KUKA KRL program: EPS_2_25716_MHCR11_A_20250905053025.src

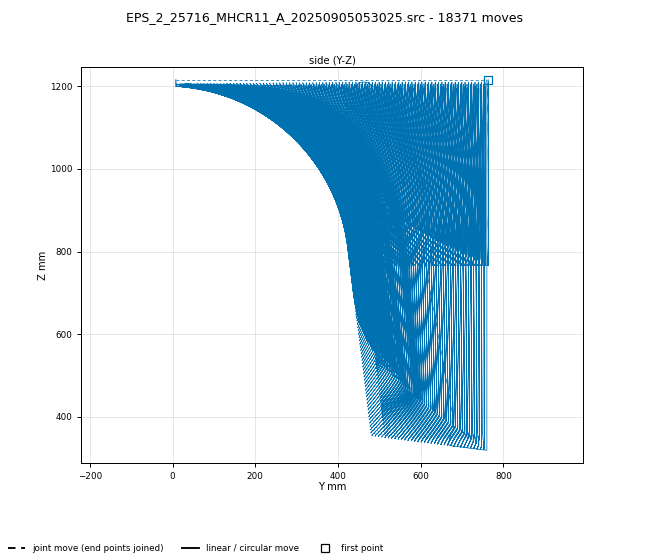
[picture p0: tool path of EPS_2_25716_MHCR11_A_20250905053025.src, 18371 of 18373 moves have a stored position in this frame; points joined in program order, loops and branches not executed]
&ACCESS RVP
&REL 4
&COMMENT QRS 19112012
&PARAM EDITMASK = *
DEF PART()
EXT BAS (BAS_COMMAND :IN,REAL :IN )
INT I
BAS (#INITMOV,0 )

;KUKA QRS Post kuka4.cps  Date:22-06-2017 !

File_ID=2809

QRS_PRE_INIT()

;Init var - Until changes are made in qrs_pre_init
Outlet_Square_prg=0
Inlet_1_Square_prg=0
Inlet_2_Square_prg=0
Inlet_3_Square_prg=0
Inlet_4_Square_prg=0
Inlet_5_Square_prg=0

Outlet_1={X 0.000, Y 457.000, Z 786.000, B 0.000, E1 0.000 }
Inlet_1={X 0.000, Y 457.000, Z 776.000, B 0.000, E1 174.000 }
Outlet_1_type=838
Inlet_1_type=838
;QRS#1=Sidecore dimensions
;QRS#2=825-33" Concrete
;QRS#3=825-33" Concrete
;QRS#4=
;QRS#5=
;QRS#6=
;QRS#7=
;QRS#8=
;QRS#9=S306-46
;QRS#10=S306-46
;QRS#11=
;QRS#12=
;QRS#13=
;QRS#14=
;QRS#15=
;QRS#16=1524x152x1676 5,5'
;QRS#17=EPS Height
;QRS#18=1205
;QRS#19=*
;QRS#20= UPDATED VERSION 22-06-2017
;QRS#21=*
Outlet_Square=0650
Inlet_1_Square=0650
Inlet_2_Square=0
Inlet_3_Square=0
Inlet_4_Square=0
Inlet_5_Square=0
Mill_Square=1
Outlet_Square_Prg=267
Inlet_1_Square_prg=267

QRS_INIT()

$ADVANCE=5

; T1
PTP {E1 176.625,E2 176.625}
PTP {X 0,Y 763.403,A -85,B 0,C 180,E1 176.625,E2 176.625,E3 0,E4 0,E5 0,E6 0}
QRS_SPEED_INIT()
LIN {X 0,Y 763.403,Z 1215,A -85,B 0,C 180,E1 176.625,E2 176.625,E3 0,E4 0,E5 0,E6 0} C_VEL
LIN {X 0,Y 763.403,Z 769.06,A -85,B 0,C 180,E1 176.625,E2 176.625} C_VEL
LIN {X 0,Y 763.516,Z 767.06,A -85,B 0,C 180,E1 176.775,E2 176.775} C_VEL
LIN {X 0,Y 763.851,Z 767.06,A -85,B 0,C 180,E1 177.187,E2 177.187} C_VEL
LIN {X 0,Y 763.775,Z 767.06,A -85,B 0,C 180,E1 184.693,E2 184.693} C_VEL
LIN {X 0,Y 763.789,Z 767.06,A -85,B 0,C 180,E1 192.281,E2 192.281} C_VEL
LIN {X 0,Y 763.833,Z 767.06,A -85,B 0,C 180,E1 200.095,E2 200.095} C_VEL
LIN {X 0,Y 763.8,Z 767.06,A -85,B 0,C 180,E1 208.326,E2 208.326} C_VEL
LIN {X 0,Y 762.389,Z 767.06,A -85,B 0,C 180,E1 210.541,E2 210.541} C_VEL
LIN {X 0,Y 762.703,Z 767.06,A -85,B 0,C 180,E1 214.993,E2 214.993} C_VEL
LIN {X 0,Y 763.704,Z 767.06,A -85,B 0,C 180,E1 216.697,E2 216.697} C_VEL
LIN {X 0,Y 763.451,Z 767.06,A -85,B 0,C 180,E1 224.739,E2 224.739} C_VEL
LIN {X 0,Y 763.703,Z 767.06,A -85,B 0,C 180,E1 225.281,E2 225.281} C_VEL
LIN {X 0,Y 763.812,Z 767.06,A -85,B 0,C 180,E1 233.406,E2 233.406} C_VEL
LIN {X 0,Y 763.419,Z 767.06,A -85,B 0,C 180,E1 233.624,E2 233.624} C_VEL
LIN {X 0,Y 763.046,Z 767.06,A -85,B 0,C 180,E1 233.668,E2 233.668} C_VEL
LIN {X 0,Y 762.775,Z 769.023,A -85,B 0,C 180,E1 233.717,E2 233.717} C_VEL
LIN {X 0,Y 763.466,Z 807.779,A -85,B 0,C 180,E1 234.197,E2 234.197} C_VEL
LIN {X 0,Y 763.742,Z 829.636,A -85,B 0,C 180,E1 234.483,E2 234.483} C_VEL
LIN {X 0,Y 763.754,Z 846.275,A -85,B 0,C 180,E1 234.748,E2 234.748} C_VEL
LIN {X 0,Y 763.618,Z 862.338,A -85,B 0,C 180,E1 235.056,E2 235.056} C_VEL
LIN {X 0,Y 763.237,Z 876.777,A -85,B 0,C 180,E1 235.362,E2 235.362} C_VEL
LIN {X 0,Y 763.626,Z 894.422,A -85,B 0,C 180,E1 235.847,E2 235.847} C_VEL
LIN {X 0,Y 763.699,Z 916.902,A -85,B 0,C 180,E1 236.542,E2 236.542} C_VEL
LIN {X 0,Y 763.604,Z 937.208,A -85,B 0,C 180,E1 237.264,E2 237.264} C_VEL
LIN {X 0,Y 763.43,Z 948.906,A -85,B 0,C 180,E1 237.721,E2 237.721} C_VEL
LIN {X 0,Y 763.574,Z 957.186,A -85,B 0,C 180,E1 238.074,E2 238.074} C_VEL
LIN {X 0,Y 763.561,Z 973.321,A -85,B 0,C 180,E1 238.795,E2 238.795} C_VEL
LIN {X 0,Y 763.553,Z 990.951,A -85,B 0,C 180,E1 239.666,E2 239.666} C_VEL
LIN {X 0,Y 763.64,Z 1008.434,A -85,B 0,C 180,E1 240.621,E2 240.621} C_VEL
LIN {X 0,Y 763.573,Z 1024.267,A -85,B 0,C 180,E1 241.555,E2 241.555} C_VEL
LIN {X 0,Y 763.324,Z 1040.379,A -85,B 0,C 180,E1 242.584,E2 242.584} C_VEL
LIN {X 0,Y 763.281,Z 1055.421,A -85,B 0,C 180,E1 243.634,E2 243.634} C_VEL
LIN {X 0,Y 763.581,Z 1070.933,A -85,B 0,C 180,E1 244.825,E2 244.825} C_VEL
LIN {X 0,Y 763.679,Z 1081.725,A -85,B 0,C 180,E1 245.706,E2 245.706} C_VEL
LIN {X 0,Y 763.252,Z 1096.523,A -85,B 0,C 180,E1 246.989,E2 246.989} C_VEL
LIN {X 0,Y 763.129,Z 1109.853,A -85,B 0,C 180,E1 248.262,E2 248.262} C_VEL
LIN {X 0,Y 763.47,Z 1121.627,A -85,B 0,C 180,E1 249.493,E2 249.493} C_VEL
LIN {X 0,Y 763.789,Z 1128.839,A -85,B 0,C 180,E1 250.312,E2 250.312} C_VEL
LIN {X 0,Y 763.599,Z 1133.682,A -85,B 0,C 180,E1 250.86,E2 250.86} C_VEL
LIN {X 0,Y 763.002,Z 1144.009,A -85,B 0,C 180,E1 252.116,E2 252.116} C_VEL
LIN {X 0,Y 762.888,Z 1154.837,A -85,B 0,C 180,E1 253.587,E2 253.587} C_VEL
LIN {X 0,Y 763.437,Z 1163.995,A -85,B 0,C 180,E1 254.972,E2 254.972} C_VEL
LIN {X 0,Y 763.849,Z 1168.884,A -85,B 0,C 180,E1 255.795,E2 255.795} C_VEL
LIN {X 0,Y 763.459,Z 1172.713,A -85,B 0,C 180,E1 256.432,E2 256.432} C_VEL
LIN {X 0,Y 762.709,Z 1180.75,A -85,B 0,C 180,E1 257.942,E2 257.942} C_VEL
LIN {X 0,Y 762.709,Z 1187.417,A -85,B 0,C 180,E1 259.378,E2 259.378} C_VEL
LIN {X 0,Y 763.283,Z 1192.233,A -85,B 0,C 180,E1 260.577,E2 260.577} C_VEL
LIN {X 0,Y 763.861,Z 1195.667,A -85,B 0,C 180,E1 261.533,E2 261.533} C_VEL
LIN {X 0,Y 763.274,Z 1198.713,A -85,B 0,C 180,E1 262.474,E2 262.474} C_VEL
LIN {X 0,Y 762.669,Z 1202.591,A -85,B 0,C 180,E1 263.886,E2 263.886} C_VEL
LIN {X 0,Y 762.823,Z 1205.612,A -85,B 0,C 180,E1 265.302,E2 265.302} C_VEL
LIN {X 0,Y 763.582,Z 1207.795,A -85,B 0,C 180,E1 266.708,E2 266.708} C_VEL
LIN {X 0,Y 763.887,Z 1208.357,A -85,B 0,C 180,E1 267.187,E2 267.187} C_VEL
LIN {X 0,Y 762.685,Z 1209.719,A -85,B 0,C 180,E1 269.062,E2 269.062} C_VEL
LIN {X 0,Y 762.503,Z 1209.722,A -85,B 0,C 180,E1 270.939,E2 270.939} C_VEL
LIN {X 0,Y 763.555,Z 1208.375,A -85,B 0,C 180,E1 272.815,E2 272.815} C_VEL
LIN {X 0,Y 763.68,Z 1207.369,A -85,B 0,C 180,E1 273.603,E2 273.603} C_VEL
LIN {X 0,Y 763.024,Z 1205.607,A -85,B 0,C 180,E1 274.698,E2 274.698} C_VEL
LIN {X 0,Y 762.624,Z 1202.589,A -85,B 0,C 180,E1 276.115,E2 276.115} C_VEL
LIN {X 0,Y 763.008,Z 1198.714,A -85,B 0,C 180,E1 277.529,E2 277.529} C_VEL
LIN {X 0,Y 763.565,Z 1195.67,A -85,B 0,C 180,E1 278.471,E2 278.471} C_VEL
LIN {X 0,Y 763.861,Z 1193.987,A -85,B 0,C 180,E1 278.942,E2 278.942} C_VEL
LIN {X 0,Y 763.295,Z 1190.396,A -85,B 0,C 180,E1 279.899,E2 279.899} C_VEL
LIN {X 0,Y 762.849,Z 1186.331,A -85,B 0,C 180,E1 280.859,E2 280.859} C_VEL
LIN {X 0,Y 762.72,Z 1179.546,A -85,B 0,C 180,E1 282.299,E2 282.299} C_VEL
LIN {X 0,Y 763.241,Z 1172.709,A -85,B 0,C 180,E1 283.573,E2 283.573} C_VEL
LIN {X 0,Y 763.817,Z 1166.178,A -85,B 0,C 180,E1 284.656,E2 284.656} C_VEL
LIN {X 0,Y 763.575,Z 1163.464,A -85,B 0,C 180,E1 285.111,E2 285.111} C_VEL
LIN {X 0,Y 762.944,Z 1153.1,A -85,B 0,C 180,E1 286.658,E2 286.658} C_VEL
LIN {X 0,Y 762.95,Z 1144.002,A -85,B 0,C 180,E1 287.886,E2 287.886} C_VEL
LIN {X 0,Y 763.507,Z 1132.817,A -85,B 0,C 180,E1 289.248,E2 289.248} C_VEL
LIN {X 0,Y 763.777,Z 1127.109,A -85,B 0,C 180,E1 289.882,E2 289.882} C_VEL
LIN {X 0,Y 763.473,Z 1119.599,A -85,B 0,C 180,E1 290.721,E2 290.721} C_VEL
LIN {X 0,Y 763.074,Z 1107.203,A -85,B 0,C 180,E1 292,E2 292} C_VEL
LIN {X 0,Y 763.142,Z 1095.102,A -85,B 0,C 180,E1 293.143,E2 293.143} C_VEL
LIN {X 0,Y 763.577,Z 1080.937,A -85,B 0,C 180,E1 294.361,E2 294.361} C_VEL
LIN {X 0,Y 763.638,Z 1069.815,A -85,B 0,C 180,E1 295.264,E2 295.264} C_VEL
LIN {X 0,Y 763.313,Z 1053.595,A -85,B 0,C 180,E1 296.496,E2 296.496} C_VEL
LIN {X 0,Y 763.281,Z 1038.391,A -85,B 0,C 180,E1 297.551,E2 297.551} C_VEL
LIN {X 0,Y 763.531,Z 1021.454,A -85,B 0,C 180,E1 298.617,E2 298.617} C_VEL
LIN {X 0,Y 763.61,Z 1005.589,A -85,B 0,C 180,E1 299.542,E2 299.542} C_VEL
LIN {X 0,Y 763.569,Z 987.905,A -85,B 0,C 180,E1 300.489,E2 300.489} C_VEL
LIN {X 0,Y 763.539,Z 970.163,A -85,B 0,C 180,E1 301.353,E2 301.353} C_VEL
LIN {X 0,Y 763.605,Z 952.774,A -85,B 0,C 180,E1 302.117,E2 302.117} C_VEL
LIN {X 0,Y 763.432,Z 938.395,A -85,B 0,C 180,E1 302.697,E2 302.697} C_VEL
LIN {X 0,Y 763.616,Z 929.2,A -85,B 0,C 180,E1 303.028,E2 303.028} C_VEL
LIN {X 0,Y 763.715,Z 913.957,A -85,B 0,C 180,E1 303.553,E2 303.553} C_VEL
LIN {X 0,Y 763.679,Z 893.472,A -85,B 0,C 180,E1 304.176,E2 304.176} C_VEL
LIN {X 0,Y 763.499,Z 875.748,A -85,B 0,C 180,E1 304.649,E2 304.649} C_VEL
LIN {X 0,Y 763.243,Z 865.606,A -85,B 0,C 180,E1 304.895,E2 304.895} C_VEL
LIN {X 0,Y 763.621,Z 848.959,A -85,B 0,C 180,E1 305.209,E2 305.209} C_VEL
LIN {X 0,Y 763.7,Z 832.013,A -85,B 0,C 180,E1 305.485,E2 305.485} C_VEL
LIN {X 0,Y 763.622,Z 816.113,A -85,B 0,C 180,E1 305.7,E2 305.7} C_VEL
LIN {X 0,Y 762.846,Z 771.116,A -85,B 0,C 180,E1 306.255,E2 306.255} C_VEL
LIN {X 0,Y 763.396,Z 767.06,A -85,B 0,C 180,E1 306.373,E2 306.373} C_VEL
LIN {X 0,Y 763.835,Z 767.06,A -85,B 0,C 180,E1 306.471,E2 306.471} C_VEL
LIN {X 0,Y 763.721,Z 767.06,A -85,B 0,C 180,E1 312.136,E2 312.136} C_VEL
LIN {X 0,Y 763.551,Z 767.06,A -85,B 0,C 180,E1 312.564,E2 312.564} C_VEL
LIN {X 0,Y 763.769,Z 767.06,A -85,B 0,C 180,E1 320.267,E2 320.267} C_VEL
LIN {X 0,Y 763.639,Z 767.06,A -85,B 0,C 180,E1 326.576,E2 326.576} C_VEL
LIN {X 0,Y 763.406,Z 767.06,A -85,B 0,C 180,E1 327.302,E2 327.302} C_VEL
LIN {X 0,Y 763.789,Z 767.06,A -85,B 0,C 180,E1 333.783,E2 333.783} C_VEL
LIN {X 0,Y 763.823,Z 767.06,A -85,B 0,C 180,E1 341.889,E2 341.889} C_VEL
LIN {X 0,Y 763.795,Z 767.06,A -85,B 0,C 180,E1 349.631,E2 349.631} C_VEL
LIN {X 0,Y 763.807,Z 767.06,A -85,B 0,C 180,E1 357.187,E2 357.187} C_VEL
LIN {X 0,Y 763.852,Z 767.06,A -85,B 0,C 180,E1 364.692,E2 364.692} C_VEL
LIN {X 0,Y 763.823,Z 767.06,A -85,B 0,C 180,E1 372.28,E2 372.28} C_VEL
LIN {X 0,Y 763.801,Z 767.06,A -85,B 0,C 180,E1 380.096,E2 380.096} C_VEL
LIN {X 0,Y 763.792,Z 767.06,A -85,B 0,C 180,E1 388.326,E2 388.326} C_VEL
LIN {X 0,Y 762.011,Z 767.06,A -85,B 0,C 180,E1 393.238,E2 393.238} C_VEL
LIN {X 0,Y 762.68,Z 767.06,A -85,B 0,C 180,E1 394.995,E2 394.995} C_VEL
LIN {X 0,Y 763.679,Z 767.06,A -85,B 0,C 180,E1 396.693,E2 396.693} C_VEL
LIN {X 0,Y 763.735,Z 767.06,A -85,B 0,C 180,E1 404.718,E2 404.718} C_VEL
LIN {X 0,Y 763.517,Z 767.06,A -85,B 0,C 180,E1 405.266,E2 405.266} C_VEL
LIN {X 0,Y 762.413,Z 767.06,A -85,B 0,C 180,E1 410.39,E2 410.39} C_VEL
LIN {X 0,Y 763.777,Z 767.06,A -85,B 0,C 180,E1 412.742,E2 412.742} C_VEL
LIN {X 0,Y 762.705,Z 767.06,A -85,B 0,C 180,E1 417.268,E2 417.268} C_VEL
LIN {X 0,Y 763.741,Z 767.06,A -85,B 0,C 180,E1 419.519,E2 419.519} C_VEL
LIN {X 0,Y 762.986,Z 767.06,A -85,B 0,C 180,E1 419.632,E2 419.632} C_VEL
LIN {X 0,Y 762.012,Z 767.06,A -85,B 0,C 180,E1 419.699,E2 419.699} C_VEL
LIN {X 0,Y 761.848,Z 768.42,A -85,B 0,C 180,E1 419.729,E2 419.729} C_VEL
LIN {X 0,Y 763.1,Z 799.119,A -85,B 0,C 180,E1 420.147,E2 420.147} C_VEL
LIN {X 0,Y 763.541,Z 819.735,A -85,B 0,C 180,E1 420.428,E2 420.428} C_VEL
LIN {X 0,Y 763.6,Z 834.791,A -85,B 0,C 180,E1 420.669,E2 420.669} C_VEL
LIN {X 0,Y 763.421,Z 851.973,A -85,B 0,C 180,E1 420.992,E2 420.992} C_VEL
LIN {X 0,Y 763.268,Z 861.057,A -85,B 0,C 180,E1 421.186,E2 421.186} C_VEL
LIN {X 0,Y 763.604,Z 877.237,A -85,B 0,C 180,E1 421.603,E2 421.603} C_VEL
LIN {X 0,Y 763.656,Z 889.927,A -85,B 0,C 180,E1 421.967,E2 421.967} C_VEL
LIN {X 0,Y 763.604,Z 907.903,A -85,B 0,C 180,E1 422.528,E2 422.528} C_VEL
LIN {X 0,Y 763.391,Z 924.777,A -85,B 0,C 180,E1 423.113,E2 423.113} C_VEL
LIN {X 0,Y 763.591,Z 944.955,A -85,B 0,C 180,E1 423.93,E2 423.93} C_VEL
LIN {X 0,Y 763.593,Z 963.795,A -85,B 0,C 180,E1 424.775,E2 424.775} C_VEL
LIN {X 0,Y 763.634,Z 981.026,A -85,B 0,C 180,E1 425.629,E2 425.629} C_VEL
LIN {X 0,Y 763.585,Z 996.993,A -85,B 0,C 180,E1 426.489,E2 426.489} C_VEL
LIN {X 0,Y 763.393,Z 1014.248,A -85,B 0,C 180,E1 427.501,E2 427.501} C_VEL
LIN {X 0,Y 763.321,Z 1030.001,A -85,B 0,C 180,E1 428.513,E2 428.513} C_VEL
LIN {X 0,Y 763.583,Z 1046.055,A -85,B 0,C 180,E1 429.648,E2 429.648} C_VEL
LIN {X 0,Y 763.634,Z 1060.068,A -85,B 0,C 180,E1 430.711,E2 430.711} C_VEL
LIN {X 0,Y 763.27,Z 1074.393,A -85,B 0,C 180,E1 431.875,E2 431.875} C_VEL
LIN {X 0,Y 763.124,Z 1086.926,A -85,B 0,C 180,E1 432.979,E2 432.979} C_VEL
LIN {X 0,Y 763.429,Z 1099.823,A -85,B 0,C 180,E1 434.223,E2 434.223} C_VEL
LIN {X 0,Y 763.747,Z 1110.439,A -85,B 0,C 180,E1 435.328,E2 435.328} C_VEL
LIN {X 0,Y 763.085,Z 1124.008,A -85,B 0,C 180,E1 436.842,E2 436.842} C_VEL
LIN {X 0,Y 762.891,Z 1134.864,A -85,B 0,C 180,E1 438.184,E2 438.184} C_VEL
LIN {X 0,Y 763.251,Z 1143.702,A -85,B 0,C 180,E1 439.385,E2 439.385} C_VEL
LIN {X 0,Y 763.85,Z 1151.677,A -85,B 0,C 180,E1 440.583,E2 440.583} C_VEL
LIN {X 0,Y 763.448,Z 1156.174,A -85,B 0,C 180,E1 441.291,E2 441.291} C_VEL
LIN {X 0,Y 762.851,Z 1163.209,A -85,B 0,C 180,E1 442.469,E2 442.469} C_VEL
LIN {X 0,Y 762.709,Z 1170.698,A -85,B 0,C 180,E1 443.886,E2 443.886} C_VEL
LIN {X 0,Y 763.298,Z 1177.26,A -85,B 0,C 180,E1 445.304,E2 445.304} C_VEL
LIN {X 0,Y 763.852,Z 1180.947,A -85,B 0,C 180,E1 446.207,E2 446.207} C_VEL
LIN {X 0,Y 763.243,Z 1184.625,A -85,B 0,C 180,E1 447.184,E2 447.184} C_VEL
LIN {X 0,Y 762.669,Z 1188.384,A -85,B 0,C 180,E1 448.309,E2 448.309} C_VEL
LIN {X 0,Y 762.548,Z 1191.547,A -85,B 0,C 180,E1 449.436,E2 449.436} C_VEL
LIN {X 0,Y 762.732,Z 1193.38,A -85,B 0,C 180,E1 450.187,E2 450.187} C_VEL
LIN {X 0,Y 763.114,Z 1194.976,A -85,B 0,C 180,E1 450.938,E2 450.938} C_VEL
LIN {X 0,Y 763.602,Z 1196.333,A -85,B 0,C 180,E1 451.688,E2 451.688} C_VEL
LIN {X 0,Y 763.324,Z 1198.172,A -85,B 0,C 180,E1 452.936,E2 452.936} C_VEL
LIN {X 0,Y 762.536,Z 1199.628,A -85,B 0,C 180,E1 454.7,E2 454.7} C_VEL
LIN {X 0,Y 762.965,Z 1199.803,A -85,B 0,C 180,E1 456.583,E2 456.583} C_VEL
LIN {X 0,Y 763.581,Z 1198.687,A -85,B 0,C 180,E1 458.47,E2 458.47} C_VEL
LIN {X 0,Y 762.998,Z 1197.578,A -85,B 0,C 180,E1 459.426,E2 459.426} C_VEL
LIN {X 0,Y 762.641,Z 1196.103,A -85,B 0,C 180,E1 460.384,E2 460.384} C_VEL
LIN {X 0,Y 762.637,Z 1194.253,A -85,B 0,C 180,E1 461.34,E2 461.34} C_VEL
LIN {X 0,Y 763.263,Z 1190.71,A -85,B 0,C 180,E1 462.789,E2 462.789} C_VEL
LIN {X 0,Y 763.555,Z 1189.344,A -85,B 0,C 180,E1 463.258,E2 463.258} C_VEL
LIN {X 0,Y 763.811,Z 1187.407,A -85,B 0,C 180,E1 463.888,E2 463.888} C_VEL
LIN {X 0,Y 763.133,Z 1183.599,A -85,B 0,C 180,E1 465.018,E2 465.018} C_VEL
LIN {X 0,Y 762.714,Z 1179.102,A -85,B 0,C 180,E1 466.173,E2 466.173} C_VEL
LIN {X 0,Y 762.716,Z 1175.906,A -85,B 0,C 180,E1 466.907,E2 466.907} C_VEL
LIN {X 0,Y 763.121,Z 1170.175,A -85,B 0,C 180,E1 468.128,E2 468.128} C_VEL
LIN {X 0,Y 763.799,Z 1163.946,A -85,B 0,C 180,E1 469.285,E2 469.285} C_VEL
LIN {X 0,Y 763.705,Z 1161.721,A -85,B 0,C 180,E1 469.692,E2 469.692} C_VEL
LIN {X 0,Y 762.997,Z 1153.575,A -85,B 0,C 180,E1 471.06,E2 471.06} C_VEL
LIN {X 0,Y 762.846,Z 1142.901,A -85,B 0,C 180,E1 472.642,E2 472.642} C_VEL
LIN {X 0,Y 763.396,Z 1132.405,A -85,B 0,C 180,E1 474.029,E2 474.029} C_VEL
LIN {X 0,Y 763.823,Z 1125.679,A -85,B 0,C 180,E1 474.844,E2 474.844} C_VEL
LIN {X 0,Y 763.591,Z 1120.756,A -85,B 0,C 180,E1 475.433,E2 475.433} C_VEL
LIN {X 0,Y 763.09,Z 1110.107,A -85,B 0,C 180,E1 476.635,E2 476.635} C_VEL
LIN {X 0,Y 762.965,Z 1098.577,A -85,B 0,C 180,E1 477.827,E2 477.827} C_VEL
LIN {X 0,Y 763.386,Z 1085.174,A -85,B 0,C 180,E1 479.084,E2 479.084} C_VEL
LIN {X 0,Y 763.705,Z 1072.505,A -85,B 0,C 180,E1 480.185,E2 480.185} C_VEL
LIN {X 0,Y 763.391,Z 1058.076,A -85,B 0,C 180,E1 481.363,E2 481.363} C_VEL
LIN {X 0,Y 763.252,Z 1043.524,A -85,B 0,C 180,E1 482.459,E2 482.459} C_VEL
LIN {X 0,Y 763.44,Z 1028.158,A -85,B 0,C 180,E1 483.514,E2 483.514} C_VEL
LIN {X 0,Y 763.564,Z 1011.608,A -85,B 0,C 180,E1 484.561,E2 484.561} C_VEL
LIN {X 0,Y 763.566,Z 995.668,A -85,B 0,C 180,E1 485.494,E2 485.494} C_VEL
LIN {X 0,Y 763.505,Z 978.376,A -85,B 0,C 180,E1 486.423,E2 486.423} C_VEL
LIN {X 0,Y 763.565,Z 961.011,A -85,B 0,C 180,E1 487.269,E2 487.269} C_VEL
LIN {X 0,Y 763.405,Z 943.665,A -85,B 0,C 180,E1 488.045,E2 488.045} C_VEL
LIN {X 0,Y 763.686,Z 922.777,A -85,B 0,C 180,E1 488.854,E2 488.854} C_VEL
LIN {X 0,Y 763.687,Z 903.938,A -85,B 0,C 180,E1 489.51,E2 489.51} C_VEL
LIN {X 0,Y 763.593,Z 883.295,A -85,B 0,C 180,E1 490.141,E2 490.141} C_VEL
LIN {X 0,Y 763.277,Z 868.309,A -85,B 0,C 180,E1 490.552,E2 490.552} C_VEL
LIN {X 0,Y 763.669,Z 851.249,A -85,B 0,C 180,E1 490.92,E2 490.92} C_VEL
LIN {X 0,Y 763.742,Z 833.97,A -85,B 0,C 180,E1 491.247,E2 491.247} C_VEL
LIN {X 0,Y 763.689,Z 817.714,A -85,B 0,C 180,E1 491.503,E2 491.503} C_VEL
LIN {X 0,Y 763.172,Z 792.315,A -85,B 0,C 180,E1 491.836,E2 491.836} C_VEL
LIN {X 0,Y 762.208,Z 767.952,A -85,B 0,C 180,E1 492.167,E2 492.167} C_VEL
LIN {X 0,Y 762.247,Z 767.06,A -85,B 0,C 180,E1 492.185,E2 492.185} C_VEL
LIN {X 0,Y 762.641,Z 767.06,A -85,B 0,C 180,E1 492.209,E2 492.209} C_VEL
LIN {X 0,Y 763.806,Z 767.06,A -85,B 0,C 180,E1 492.37,E2 492.37} C_VEL
LIN {X 0,Y 763.814,Z 767.06,A -85,B 0,C 180,E1 494.71,E2 494.71} C_VEL
LIN {X 0,Y 763.513,Z 767.06,A -85,B 0,C 180,E1 495.266,E2 495.266} C_VEL
LIN {X 0,Y 762.427,Z 767.06,A -85,B 0,C 180,E1 500.387,E2 500.387} C_VEL
LIN {X 0,Y 763.796,Z 767.06,A -85,B 0,C 180,E1 502.743,E2 502.743} C_VEL
LIN {X 0,Y 763.654,Z 767.06,A -85,B 0,C 180,E1 510.149,E2 510.149} C_VEL
LIN {X 0,Y 762.937,Z 767.06,A -85,B 0,C 180,E1 511.639,E2 511.639} C_VEL
LIN {X 0,Y 763.766,Z 767.06,A -85,B 0,C 180,E1 517.893,E2 517.893} C_VEL
LIN {X 0,Y 763.499,Z 767.06,A -85,B 0,C 180,E1 524.951,E2 524.951} C_VEL
LIN {X 0,Y 763.691,Z 767.06,A -85,B 0,C 180,E1 525.791,E2 525.791} C_VEL
LIN {X 0,Y 763.843,Z 767.06,A -85,B 0,C 180,E1 529.632,E2 529.632} C_VEL
LIN {X 0,Y 763.516,Z 767.06,A -85,B 0,C 180,E1 536.775,E2 536.775} C_VEL
LIN {X 0,Y 754.474,Z 767.06,A -85,B 0,C 180,E1 539.373,E2 539.373} C_VEL
LIN {X 0,Y 754.654,Z 767.06,A -85,B 0,C 180,E1 546.335,E2 546.335} C_VEL
LIN {X 0,Y 754.949,Z 767.06,A -85,B 0,C 180,E1 553.348,E2 553.348} C_VEL
LIN {X 0,Y 755.086,Z 767.06,A -85,B 0,C 180,E1 560.949,E2 560.949} C_VEL
LIN {X 0,Y 754.927,Z 767.06,A -85,B 0,C 180,E1 569.477,E2 569.477} C_VEL
LIN {X 0,Y 754.776,Z 767.06,A -85,B 0,C 180,E1 577.789,E2 577.789} C_VEL
LIN {X 0,Y 754.997,Z 767.06,A -85,B 0,C 180,E1 586.133,E2 586.133} C_VEL
LIN {X 0,Y 755.979,Z 769.043,A -85,B 0,C 180,E1 593.339,E2 593.339} C_VEL
LIN {X 0,Y 756.783,Z 872.028,A -85,B 0,C 180,E1 594.912,E2 594.912} C_VEL
LIN {X 0,Y 756.488,Z 949.209,A -85,B 0,C 180,E1 597.4,E2 597.4} C_VEL
LIN {X 0,Y 756.272,Z 1019.819,A -85,B 0,C 180,E1 600.986,E2 600.986} C_VEL
LIN {X 0,Y 756.024,Z 1082.268,A -85,B 0,C 180,E1 605.489,E2 605.489} C_VEL
LIN {X 0,Y 755.719,Z 1134.991,A -85,B 0,C 180,E1 610.815,E2 610.815} C_VEL
LIN {X 0,Y 755.547,Z 1173.024,A -85,B 0,C 180,E1 616.346,E2 616.346} C_VEL
LIN {X 0,Y 755.267,Z 1199.02,A -85,B 0,C 180,E1 622.499,E2 622.499} C_VEL
LIN {X 0,Y 755.109,Z 1209.402,A -85,B 0,C 180,E1 628.272,E2 628.272} C_VEL
LIN {X 0,Y 755.402,Z 1206.834,A -85,B 0,C 180,E1 634.027,E2 634.027} C_VEL
LIN {X 0,Y 755.214,Z 1189.941,A -85,B 0,C 180,E1 640.118,E2 640.118} C_VEL
LIN {X 0,Y 755.342,Z 1160.518,A -85,B 0,C 180,E1 645.724,E2 645.724} C_VEL
LIN {X 0,Y 755.517,Z 1116.643,A -85,B 0,C 180,E1 651.258,E2 651.258} C_VEL
LIN {X 0,Y 755.832,Z 1059.275,A -85,B 0,C 180,E1 656.351,E2 656.351} C_VEL
LIN {X 0,Y 756.399,Z 992.307,A -85,B 0,C 180,E1 660.577,E2 660.577} C_VEL
LIN {X 0,Y 756.847,Z 920.414,A -85,B 0,C 180,E1 663.676,E2 663.676} C_VEL
LIN {X 0,Y 757.101,Z 846.686,A -85,B 0,C 180,E1 665.601,E2 665.601} C_VEL
LIN {X 0,Y 755.663,Z 767.06,A -85,B 0,C 180,E1 666.739,E2 666.739} C_VEL
LIN {X 0,Y 754.628,Z 767.06,A -85,B 0,C 180,E1 673.889,E2 673.889} C_VEL
LIN {X 0,Y 755.408,Z 767.06,A -85,B 0,C 180,E1 680.779,E2 680.779} C_VEL
LIN {X 0,Y 755.067,Z 767.06,A -85,B 0,C 180,E1 687.849,E2 687.849} C_VEL
LIN {X 0,Y 755.237,Z 767.06,A -85,B 0,C 180,E1 694.43,E2 694.43} C_VEL
LIN {X 0,Y 754.909,Z 767.06,A -85,B 0,C 180,E1 703.073,E2 703.073} C_VEL
LIN {X 0,Y 755.337,Z 767.06,A -85,B 0,C 180,E1 710.183,E2 710.183} C_VEL
LIN {X 0,Y 754.992,Z 767.06,A -85,B 0,C 180,E1 718.285,E2 718.285} C_VEL
LIN {X 0,Y 754.857,Z 767.06,A -85,B 0,C 180,E1 726.071,E2 726.071} C_VEL
LIN {X 0,Y 754.97,Z 767.06,A -85,B 0,C 180,E1 733.371,E2 733.371} C_VEL
LIN {X 0,Y 755.059,Z 767.06,A -85,B 0,C 180,E1 740.953,E2 740.953} C_VEL
LIN {X 0,Y 754.845,Z 767.06,A -85,B 0,C 180,E1 749.507,E2 749.507} C_VEL
LIN {X 0,Y 754.782,Z 767.06,A -85,B 0,C 180,E1 757.817,E2 757.817} C_VEL
LIN {X 0,Y 754.895,Z 767.06,A -85,B 0,C 180,E1 766.131,E2 766.131} C_VEL
LIN {X 0,Y 755.173,Z 767.06,A -85,B 0,C 180,E1 773.675,E2 773.675} C_VEL
LIN {X 0,Y 755.556,Z 767.06,A -85,B 0,C 180,E1 779.343,E2 779.343} C_VEL
LIN {X 0,Y 756.733,Z 865.954,A -85,B 0,C 180,E1 780.956,E2 780.956} C_VEL
LIN {X 0,Y 756.581,Z 941.104,A -85,B 0,C 180,E1 783.436,E2 783.436} C_VEL
LIN {X 0,Y 756.086,Z 1013.204,A -85,B 0,C 180,E1 787.135,E2 787.135} C_VEL
LIN {X 0,Y 755.601,Z 1075.643,A -85,B 0,C 180,E1 791.726,E2 791.726} C_VEL
LIN {X 0,Y 755.209,Z 1125.549,A -85,B 0,C 180,E1 796.826,E2 796.826} C_VEL
LIN {X 0,Y 754.991,Z 1162.599,A -85,B 0,C 180,E1 802.21,E2 802.21} C_VEL
LIN {X 0,Y 754.943,Z 1186.693,A -85,B 0,C 180,E1 807.699,E2 807.699} C_VEL
LIN {X 0,Y 755.341,Z 1198.166,A -85,B 0,C 180,E1 812.879,E2 812.879} C_VEL
LIN {X 0,Y 755.453,Z 1198.555,A -85,B 0,C 180,E1 818.661,E2 818.661} C_VEL
LIN {X 0,Y 755.243,Z 1184.571,A -85,B 0,C 180,E1 824.835,E2 824.835} C_VEL
LIN {X 0,Y 755.255,Z 1157.414,A -85,B 0,C 180,E1 830.573,E2 830.573} C_VEL
LIN {X 0,Y 755.499,Z 1117.265,A -85,B 0,C 180,E1 836.047,E2 836.047} C_VEL
LIN {X 0,Y 755.829,Z 1063.478,A -85,B 0,C 180,E1 841.197,E2 841.197} C_VEL
LIN {X 0,Y 756.3,Z 999.137,A -85,B 0,C 180,E1 845.606,E2 845.606} C_VEL
LIN {X 0,Y 756.75,Z 927.722,A -85,B 0,C 180,E1 849.004,E2 849.004} C_VEL
LIN {X 0,Y 757.025,Z 854.459,A -85,B 0,C 180,E1 851.204,E2 851.204} C_VEL
LIN {X 0,Y 755.775,Z 767.06,A -85,B 0,C 180,E1 852.628,E2 852.628} C_VEL
LIN {X 0,Y 755.555,Z 767.06,A -85,B 0,C 180,E1 862.45,E2 862.45} C_VEL
LIN {X 0,Y 754.854,Z 767.06,A -85,B 0,C 180,E1 871.808,E2 871.808} C_VEL
LIN {X 0,Y 754.733,Z 767.06,A -85,B 0,C 180,E1 879.396,E2 879.396} C_VEL
LIN {X 0,Y 755.395,Z 767.06,A -85,B 0,C 180,E1 886.822,E2 886.822} C_VEL
LIN {X 0,Y 754.208,Z 767.06,A -85,B 0,C 180,E1 893.638,E2 893.638} C_VEL
LIN {X 0,Y 755.053,Z 767.06,A -85,B 0,C 180,E1 898.262,E2 898.262} C_VEL
LIN {X 0,Y 754.474,Z 767.06,A -85,B 0,C 180,E1 899.373,E2 899.373} C_VEL
LIN {X 0,Y 746.33,Z 767.06,A -85,B 0,C 180,E1 902.004,E2 902.004} C_VEL
LIN {X 0,Y 746.203,Z 767.06,A -85,B 0,C 180,E1 907.581,E2 907.581} C_VEL
LIN {X 0,Y 746.85,Z 767.06,A -85,B 0,C 180,E1 913.495,E2 913.495} C_VEL
LIN {X 0,Y 747.196,Z 767.06,A -85,B 0,C 180,E1 920.797,E2 920.797} C_VEL
LIN {X 0,Y 747.459,Z 767.06,A -85,B 0,C 180,E1 928.47,E2 928.47} C_VEL
LIN {X 0,Y 747.238,Z 767.06,A -85,B 0,C 180,E1 936.772,E2 936.772} C_VEL
LIN {X 0,Y 747.003,Z 767.06,A -85,B 0,C 180,E1 946.109,E2 946.109} C_VEL
LIN {X 0,Y 747.508,Z 768.844,A -85,B 0,C 180,E1 952.851,E2 952.851} C_VEL
LIN {X 0,Y 750.106,Z 782.699,A -85,B 0,C 180,E1 953.164,E2 953.164} C_VEL
LIN {X 0,Y 750.08,Z 875.698,A -85,B 0,C 180,E1 954.638,E2 954.638} C_VEL
LIN {X 0,Y 749.523,Z 953.639,A -85,B 0,C 180,E1 957.241,E2 957.241} C_VEL
LIN {X 0,Y 748.914,Z 1024.39,A -85,B 0,C 180,E1 960.954,E2 960.954} C_VEL
LIN {X 0,Y 748.332,Z 1085.959,A -85,B 0,C 180,E1 965.549,E2 965.549} C_VEL
LIN {X 0,Y 747.758,Z 1137.766,A -85,B 0,C 180,E1 970.952,E2 970.952} C_VEL
LIN {X 0,Y 747.448,Z 1174.643,A -85,B 0,C 180,E1 976.506,E2 976.506} C_VEL
LIN {X 0,Y 747.304,Z 1199.02,A -85,B 0,C 180,E1 982.419,E2 982.419} C_VEL
LIN {X 0,Y 747.114,Z 1209.402,A -85,B 0,C 180,E1 988.254,E2 988.254} C_VEL
LIN {X 0,Y 747.384,Z 1206.834,A -85,B 0,C 180,E1 994.071,E2 994.071} C_VEL
LIN {X 0,Y 747.227,Z 1190.236,A -85,B 0,C 180,E1 1000.154,E2 1000.154} C_VEL
LIN {X 0,Y 747.355,Z 1160.52,A -85,B 0,C 180,E1 1005.896,E2 1005.896} C_VEL
LIN {X 0,Y 747.688,Z 1116.882,A -85,B 0,C 180,E1 1011.467,E2 1011.467} C_VEL
LIN {X 0,Y 748.306,Z 1061.049,A -85,B 0,C 180,E1 1016.5,E2 1016.5} C_VEL
LIN {X 0,Y 749.205,Z 994.733,A -85,B 0,C 180,E1 1020.768,E2 1020.768} C_VEL
LIN {X 0,Y 749.989,Z 923.555,A -85,B 0,C 180,E1 1023.912,E2 1023.912} C_VEL
LIN {X 0,Y 750.517,Z 849.589,A -85,B 0,C 180,E1 1025.906,E2 1025.906} C_VEL
LIN {X 0,Y 748.279,Z 770.571,A -85,B 0,C 180,E1 1027.084,E2 1027.084} C_VEL
LIN {X 0,Y 747.331,Z 767.06,A -85,B 0,C 180,E1 1027.326,E2 1027.326} C_VEL
LIN {X 0,Y 746.637,Z 767.06,A -85,B 0,C 180,E1 1033.862,E2 1033.862} C_VEL
LIN {X 0,Y 746.904,Z 767.06,A -85,B 0,C 180,E1 1041.742,E2 1041.742} C_VEL
LIN {X 0,Y 746.639,Z 767.06,A -85,B 0,C 180,E1 1048.812,E2 1048.812} C_VEL
LIN {X 0,Y 746.57,Z 767.06,A -85,B 0,C 180,E1 1055.398,E2 1055.398} C_VEL
LIN {X 0,Y 747.027,Z 767.06,A -85,B 0,C 180,E1 1062.889,E2 1062.889} C_VEL
LIN {X 0,Y 747.321,Z 767.06,A -85,B 0,C 180,E1 1070.077,E2 1070.077} C_VEL
LIN {X 0,Y 746.996,Z 767.06,A -85,B 0,C 180,E1 1078.266,E2 1078.266} C_VEL
LIN {X 0,Y 747.4,Z 767.06,A -85,B 0,C 180,E1 1085.252,E2 1085.252} C_VEL
LIN {X 0,Y 746.869,Z 767.06,A -85,B 0,C 180,E1 1093.519,E2 1093.519} C_VEL
LIN {X 0,Y 747.156,Z 767.06,A -85,B 0,C 180,E1 1100.823,E2 1100.823} C_VEL
LIN {X 0,Y 747.432,Z 767.06,A -85,B 0,C 180,E1 1108.497,E2 1108.497} C_VEL
LIN {X 0,Y 747.201,Z 767.06,A -85,B 0,C 180,E1 1116.803,E2 1116.803} C_VEL
LIN {X 0,Y 747.276,Z 767.06,A -85,B 0,C 180,E1 1125.566,E2 1125.566} C_VEL
LIN {X 0,Y 747.272,Z 767.06,A -85,B 0,C 180,E1 1133.321,E2 1133.321} C_VEL
LIN {X 0,Y 747.518,Z 768.68,A -85,B 0,C 180,E1 1138.923,E2 1138.923} C_VEL
LIN {X 0,Y 750.03,Z 863.027,A -85,B 0,C 180,E1 1140.527,E2 1140.527} C_VEL
LIN {X 0,Y 749.597,Z 938.927,A -85,B 0,C 180,E1 1143.007,E2 1143.007} C_VEL
LIN {X 0,Y 748.834,Z 1009.897,A -85,B 0,C 180,E1 1146.629,E2 1146.629} C_VEL
LIN {X 0,Y 748.124,Z 1073.156,A -85,B 0,C 180,E1 1151.244,E2 1151.244} C_VEL
LIN {X 0,Y 747.45,Z 1124.675,A -85,B 0,C 180,E1 1156.509,E2 1156.509} C_VEL
LIN {X 0,Y 747.066,Z 1162.941,A -85,B 0,C 180,E1 1162.126,E2 1162.126} C_VEL
LIN {X 0,Y 746.964,Z 1186.895,A -85,B 0,C 180,E1 1167.675,E2 1167.675} C_VEL
LIN {X 0,Y 747.333,Z 1198.236,A -85,B 0,C 180,E1 1172.909,E2 1172.909} C_VEL
LIN {X 0,Y 747.384,Z 1198.488,A -85,B 0,C 180,E1 1178.755,E2 1178.755} C_VEL
LIN {X 0,Y 747.324,Z 1185.384,A -85,B 0,C 180,E1 1184.695,E2 1184.695} C_VEL
LIN {X 0,Y 747.368,Z 1158.833,A -85,B 0,C 180,E1 1190.49,E2 1190.49} C_VEL
LIN {X 0,Y 747.633,Z 1117.632,A -85,B 0,C 180,E1 1196.226,E2 1196.226} C_VEL
LIN {X 0,Y 748.224,Z 1064.307,A -85,B 0,C 180,E1 1201.402,E2 1201.402} C_VEL
LIN {X 0,Y 749.024,Z 999.531,A -85,B 0,C 180,E1 1205.899,E2 1205.899} C_VEL
LIN {X 0,Y 749.864,Z 928.256,A -85,B 0,C 180,E1 1209.326,E2 1209.326} C_VEL
LIN {X 0,Y 750.468,Z 853.672,A -85,B 0,C 180,E1 1211.576,E2 1211.576} C_VEL
LIN {X 0,Y 747.708,Z 767.06,A -85,B 0,C 180,E1 1213.009,E2 1213.009} C_VEL
LIN {X 0,Y 747.214,Z 767.06,A -85,B 0,C 180,E1 1223.29,E2 1223.29} C_VEL
LIN {X 0,Y 746.739,Z 767.06,A -85,B 0,C 180,E1 1232.057,E2 1232.057} C_VEL
LIN {X 0,Y 746.872,Z 767.06,A -85,B 0,C 180,E1 1239.169,E2 1239.169} C_VEL
LIN {X 0,Y 747.369,Z 767.06,A -85,B 0,C 180,E1 1247.684,E2 1247.684} C_VEL
LIN {X 0,Y 747.752,Z 767.06,A -85,B 0,C 180,E1 1257.081,E2 1257.081} C_VEL
LIN {X 0,Y 746.33,Z 767.06,A -85,B 0,C 180,E1 1262.004,E2 1262.004} C_VEL
LIN {X 0,Y 739.237,Z 767.06,A -85,B 0,C 180,E1 1264.685,E2 1264.685} C_VEL
LIN {X 0,Y 738.786,Z 767.06,A -85,B 0,C 180,E1 1273.645,E2 1273.645} C_VEL
LIN {X 0,Y 739.027,Z 767.06,A -85,B 0,C 180,E1 1281.038,E2 1281.038} C_VEL
LIN {X 0,Y 738.971,Z 767.06,A -85,B 0,C 180,E1 1289.287,E2 1289.287} C_VEL
LIN {X 0,Y 738.674,Z 767.06,A -85,B 0,C 180,E1 1297.776,E2 1297.776} C_VEL
LIN {X 0,Y 738.727,Z 767.06,A -85,B 0,C 180,E1 1306.55,E2 1306.55} C_VEL
LIN {X 0,Y 739.062,Z 768.583,A -85,B 0,C 180,E1 1312.35,E2 1312.35} C_VEL
LIN {X 0,Y 743.676,Z 781.949,A -85,B 0,C 180,E1 1312.783,E2 1312.783} C_VEL
LIN {X 0,Y 743.533,Z 875.159,A -85,B 0,C 180,E1 1314.266,E2 1314.266} C_VEL
LIN {X 0,Y 742.612,Z 951.974,A -85,B 0,C 180,E1 1316.827,E2 1316.827} C_VEL
LIN {X 0,Y 741.625,Z 1023.533,A -85,B 0,C 180,E1 1320.584,E2 1320.584} C_VEL
LIN {X 0,Y 740.731,Z 1084.887,A -85,B 0,C 180,E1 1325.183,E2 1325.183} C_VEL
LIN {X 0,Y 740.056,Z 1136.557,A -85,B 0,C 180,E1 1330.592,E2 1330.592} C_VEL
LIN {X 0,Y 739.443,Z 1175.692,A -85,B 0,C 180,E1 1336.56,E2 1336.56} C_VEL
LIN {X 0,Y 739.359,Z 1199.02,A -85,B 0,C 180,E1 1342.337,E2 1342.337} C_VEL
LIN {X 0,Y 739.118,Z 1209.402,A -85,B 0,C 180,E1 1348.235,E2 1348.235} C_VEL
LIN {X 0,Y 739.35,Z 1206.834,A -85,B 0,C 180,E1 1354.115,E2 1354.115} C_VEL
LIN {X 0,Y 739.176,Z 1190.233,A -85,B 0,C 180,E1 1360.266,E2 1360.266} C_VEL
LIN {X 0,Y 739.376,Z 1160.521,A -85,B 0,C 180,E1 1366.073,E2 1366.073} C_VEL
LIN {X 0,Y 739.867,Z 1117.141,A -85,B 0,C 180,E1 1371.677,E2 1371.677} C_VEL
LIN {X 0,Y 740.737,Z 1060.479,A -85,B 0,C 180,E1 1376.837,E2 1376.837} C_VEL
LIN {X 0,Y 742.031,Z 995.01,A -85,B 0,C 180,E1 1381.083,E2 1381.083} C_VEL
LIN {X 0,Y 743.192,Z 923.447,A -85,B 0,C 180,E1 1384.269,E2 1384.269} C_VEL
LIN {X 0,Y 744.008,Z 849.51,A -85,B 0,C 180,E1 1386.272,E2 1386.272} C_VEL
LIN {X 0,Y 741.831,Z 772.891,A -85,B 0,C 180,E1 1387.433,E2 1387.433} C_VEL
LIN {X 0,Y 739.128,Z 767.06,A -85,B 0,C 180,E1 1387.824,E2 1387.824} C_VEL
LIN {X 0,Y 738.896,Z 767.06,A -85,B 0,C 180,E1 1393.433,E2 1393.433} C_VEL
LIN {X 0,Y 739.093,Z 767.06,A -85,B 0,C 180,E1 1401.262,E2 1401.262} C_VEL
LIN {X 0,Y 738.77,Z 767.06,A -85,B 0,C 180,E1 1408.442,E2 1408.442} C_VEL
LIN {X 0,Y 738.737,Z 767.06,A -85,B 0,C 180,E1 1415.12,E2 1415.12} C_VEL
LIN {X 0,Y 739.096,Z 767.06,A -85,B 0,C 180,E1 1422.7,E2 1422.7} C_VEL
LIN {X 0,Y 738.753,Z 767.06,A -85,B 0,C 180,E1 1431.153,E2 1431.153} C_VEL
LIN {X 0,Y 738.999,Z 767.06,A -85,B 0,C 180,E1 1438.247,E2 1438.247} C_VEL
LIN {X 0,Y 739.099,Z 767.06,A -85,B 0,C 180,E1 1445.688,E2 1445.688} C_VEL
LIN {X 0,Y 738.805,Z 767.06,A -85,B 0,C 180,E1 1453.669,E2 1453.669} C_VEL
LIN {X 0,Y 738.969,Z 767.06,A -85,B 0,C 180,E1 1461.065,E2 1461.065} C_VEL
LIN {X 0,Y 738.935,Z 767.06,A -85,B 0,C 180,E1 1469.289,E2 1469.289} C_VEL
LIN {X 0,Y 738.695,Z 767.06,A -85,B 0,C 180,E1 1477.784,E2 1477.784} C_VEL
LIN {X 0,Y 739.346,Z 767.06,A -85,B 0,C 180,E1 1485.074,E2 1485.074} C_VEL
LIN {X 0,Y 738.902,Z 767.06,A -85,B 0,C 180,E1 1494.206,E2 1494.206} C_VEL
LIN {X 0,Y 739.274,Z 768.666,A -85,B 0,C 180,E1 1498.439,E2 1498.439} C_VEL
LIN {X 0,Y 743.016,Z 783.088,A -85,B 0,C 180,E1 1498.832,E2 1498.832} C_VEL
LIN {X 0,Y 743.481,Z 870.987,A -85,B 0,C 180,E1 1500.37,E2 1500.37} C_VEL
LIN {X 0,Y 742.656,Z 946.965,A -85,B 0,C 180,E1 1503.007,E2 1503.007} C_VEL
LIN {X 0,Y 741.388,Z 1016.839,A -85,B 0,C 180,E1 1506.749,E2 1506.749} C_VEL
LIN {X 0,Y 740.283,Z 1078.902,A -85,B 0,C 180,E1 1511.489,E2 1511.489} C_VEL
LIN {X 0,Y 739.477,Z 1128.61,A -85,B 0,C 180,E1 1516.792,E2 1516.792} C_VEL
LIN {X 0,Y 739.158,Z 1163.282,A -85,B 0,C 180,E1 1522.042,E2 1522.042} C_VEL
LIN {X 0,Y 738.98,Z 1187.097,A -85,B 0,C 180,E1 1527.65,E2 1527.65} C_VEL
LIN {X 0,Y 739.304,Z 1198.301,A -85,B 0,C 180,E1 1532.941,E2 1532.941} C_VEL
LIN {X 0,Y 739.336,Z 1198.421,A -85,B 0,C 180,E1 1538.851,E2 1538.851} C_VEL
LIN {X 0,Y 739.25,Z 1185.151,A -85,B 0,C 180,E1 1544.859,E2 1544.859} C_VEL
LIN {X 0,Y 739.369,Z 1158.735,A -85,B 0,C 180,E1 1550.668,E2 1550.668} C_VEL
LIN {X 0,Y 739.797,Z 1118.742,A -85,B 0,C 180,E1 1556.321,E2 1556.321} C_VEL
LIN {X 0,Y 740.594,Z 1064.626,A -85,B 0,C 180,E1 1561.657,E2 1561.657} C_VEL
LIN {X 0,Y 741.763,Z 1000.643,A -85,B 0,C 180,E1 1566.155,E2 1566.155} C_VEL
LIN {X 0,Y 742.979,Z 929.799,A -85,B 0,C 180,E1 1569.612,E2 1569.612} C_VEL
LIN {X 0,Y 743.869,Z 856.128,A -85,B 0,C 180,E1 1571.885,E2 1571.885} C_VEL
LIN {X 0,Y 741.448,Z 772.05,A -85,B 0,C 180,E1 1573.302,E2 1573.302} C_VEL
LIN {X 0,Y 739.676,Z 767.06,A -85,B 0,C 180,E1 1573.611,E2 1573.611} C_VEL
LIN {X 0,Y 739.115,Z 767.06,A -85,B 0,C 180,E1 1582.726,E2 1582.726} C_VEL
LIN {X 0,Y 739.007,Z 767.06,A -85,B 0,C 180,E1 1591.147,E2 1591.147} C_VEL
LIN {X 0,Y 738.918,Z 767.06,A -85,B 0,C 180,E1 1599.037,E2 1599.037} C_VEL
LIN {X 0,Y 739.363,Z 767.06,A -85,B 0,C 180,E1 1607.548,E2 1607.548} C_VEL
LIN {X 0,Y 739.711,Z 767.06,A -85,B 0,C 180,E1 1617.05,E2 1617.05} C_VEL
LIN {X 0,Y 739.237,Z 767.06,A -85,B 0,C 180,E1 1624.685,E2 1624.685} C_VEL
LIN {X 0,Y 730.258,Z 767.06,A -85,B 0,C 180,E1 1627.364,E2 1627.364} C_VEL
LIN {X 0,Y 730.696,Z 767.06,A -85,B 0,C 180,E1 1633.799,E2 1633.799} C_VEL
LIN {X 0,Y 730.85,Z 767.06,A -85,B 0,C 180,E1 1641.285,E2 1641.285} C_VEL
LIN {X 0,Y 731.046,Z 767.06,A -85,B 0,C 180,E1 1649.17,E2 1649.17} C_VEL
LIN {X 0,Y 730.705,Z 767.06,A -85,B 0,C 180,E1 1657.747,E2 1657.747} C_VEL
LIN {X 0,Y 730.882,Z 767.06,A -85,B 0,C 180,E1 1665.965,E2 1665.965} C_VEL
LIN {X 0,Y 730.82,Z 768.902,A -85,B 0,C 180,E1 1671.854,E2 1671.854} C_VEL
LIN {X 0,Y 737.31,Z 783.467,A -85,B 0,C 180,E1 1672.425,E2 1672.425} C_VEL
LIN {X 0,Y 736.94,Z 876.7,A -85,B 0,C 180,E1 1673.936,E2 1673.936} C_VEL
LIN {X 0,Y 735.665,Z 954.209,A -85,B 0,C 180,E1 1676.57,E2 1676.57} C_VEL
LIN {X 0,Y 734.286,Z 1025.302,A -85,B 0,C 180,E1 1680.38,E2 1680.38} C_VEL
LIN {X 0,Y 733.085,Z 1086.613,A -85,B 0,C 180,E1 1685.066,E2 1685.066} C_VEL
LIN {X 0,Y 732.237,Z 1137.125,A -85,B 0,C 180,E1 1690.449,E2 1690.449} C_VEL
LIN {X 0,Y 731.674,Z 1174.646,A -85,B 0,C 180,E1 1696.209,E2 1696.209} C_VEL
LIN {X 0,Y 731.395,Z 1199.02,A -85,B 0,C 180,E1 1702.253,E2 1702.253} C_VEL
LIN {X 0,Y 731.149,Z 1209.402,A -85,B 0,C 180,E1 1708.215,E2 1708.215} C_VEL
LIN {X 0,Y 731.321,Z 1206.834,A -85,B 0,C 180,E1 1714.16,E2 1714.16} C_VEL
LIN {X 0,Y 731.257,Z 1191.083,A -85,B 0,C 180,E1 1720.151,E2 1720.151} C_VEL
LIN {X 0,Y 731.484,Z 1161.906,A -85,B 0,C 180,E1 1726.035,E2 1726.035} C_VEL
LIN {X 0,Y 732.097,Z 1118.511,A -85,B 0,C 180,E1 1731.771,E2 1731.771} C_VEL
LIN {X 0,Y 733.218,Z 1061.995,A -85,B 0,C 180,E1 1737.014,E2 1737.014} C_VEL
LIN {X 0,Y 734.896,Z 994.967,A -85,B 0,C 180,E1 1741.422,E2 1741.422} C_VEL
LIN {X 0,Y 736.446,Z 923.451,A -85,B 0,C 180,E1 1744.627,E2 1744.627} C_VEL
LIN {X 0,Y 737.5,Z 850.775,A -85,B 0,C 180,E1 1746.618,E2 1746.618} C_VEL
LIN {X 0,Y 735.661,Z 777.075,A -85,B 0,C 180,E1 1747.751,E2 1747.751} C_VEL
LIN {X 0,Y 730.997,Z 767.06,A -85,B 0,C 180,E1 1748.308,E2 1748.308} C_VEL
LIN {X 0,Y 730.437,Z 767.06,A -85,B 0,C 180,E1 1754.256,E2 1754.256} C_VEL
LIN {X 0,Y 730.769,Z 767.06,A -85,B 0,C 180,E1 1762.257,E2 1762.257} C_VEL
LIN {X 0,Y 730.857,Z 767.06,A -85,B 0,C 180,E1 1768.06,E2 1768.06} C_VEL
LIN {X 0,Y 730.806,Z 767.06,A -85,B 0,C 180,E1 1774.831,E2 1774.831} C_VEL
LIN {X 0,Y 731.177,Z 767.06,A -85,B 0,C 180,E1 1782.506,E2 1782.506} C_VEL
LIN {X 0,Y 730.785,Z 767.06,A -85,B 0,C 180,E1 1791.056,E2 1791.056} C_VEL
LIN {X 0,Y 731.033,Z 767.06,A -85,B 0,C 180,E1 1798.228,E2 1798.228} C_VEL
LIN {X 0,Y 731.3,Z 767.06,A -85,B 0,C 180,E1 1805.368,E2 1805.368} C_VEL
LIN {X 0,Y 730.714,Z 767.06,A -85,B 0,C 180,E1 1813.823,E2 1813.823} C_VEL
LIN {X 0,Y 730.799,Z 767.06,A -85,B 0,C 180,E1 1821.312,E2 1821.312} C_VEL
LIN {X 0,Y 731.005,Z 767.06,A -85,B 0,C 180,E1 1829.199,E2 1829.199} C_VEL
LIN {X 0,Y 730.723,Z 767.06,A -85,B 0,C 180,E1 1837.776,E2 1837.776} C_VEL
LIN {X 0,Y 730.869,Z 767.06,A -85,B 0,C 180,E1 1845.969,E2 1845.969} C_VEL
LIN {X 0,Y 730.959,Z 767.06,A -85,B 0,C 180,E1 1853.755,E2 1853.755} C_VEL
LIN {X 0,Y 731.165,Z 769.07,A -85,B 0,C 180,E1 1857.955,E2 1857.955} C_VEL
LIN {X 0,Y 736.561,Z 781.909,A -85,B 0,C 180,E1 1858.437,E2 1858.437} C_VEL
LIN {X 0,Y 736.858,Z 870.675,A -85,B 0,C 180,E1 1859.992,E2 1859.992} C_VEL
LIN {X 0,Y 735.714,Z 945.886,A -85,B 0,C 180,E1 1862.606,E2 1862.606} C_VEL
LIN {X 0,Y 734.154,Z 1015.744,A -85,B 0,C 180,E1 1866.359,E2 1866.359} C_VEL
LIN {X 0,Y 732.734,Z 1078.339,A -85,B 0,C 180,E1 1871.168,E2 1871.168} C_VEL
LIN {X 0,Y 731.638,Z 1128.594,A -85,B 0,C 180,E1 1876.576,E2 1876.576} C_VEL
LIN {X 0,Y 731.238,Z 1163.625,A -85,B 0,C 180,E1 1881.955,E2 1881.955} C_VEL
LIN {X 0,Y 731.01,Z 1187.298,A -85,B 0,C 180,E1 1887.624,E2 1887.624} C_VEL
LIN {X 0,Y 731.289,Z 1198.367,A -85,B 0,C 180,E1 1892.973,E2 1892.973} C_VEL
LIN {X 0,Y 731.271,Z 1198.354,A -85,B 0,C 180,E1 1898.949,E2 1898.949} C_VEL
LIN {X 0,Y 731.198,Z 1184.92,A -85,B 0,C 180,E1 1905.027,E2 1905.027} C_VEL
LIN {X 0,Y 731.366,Z 1158.219,A -85,B 0,C 180,E1 1910.923,E2 1910.923} C_VEL
LIN {X 0,Y 731.918,Z 1118.278,A -85,B 0,C 180,E1 1916.605,E2 1916.605} C_VEL
LIN {X 0,Y 733.046,Z 1064.061,A -85,B 0,C 180,E1 1921.989,E2 1921.989} C_VEL
LIN {X 0,Y 734.595,Z 1000.172,A -85,B 0,C 180,E1 1926.51,E2 1926.51} C_VEL
LIN {X 0,Y 736.141,Z 929.75,A -85,B 0,C 180,E1 1929.969,E2 1929.969} C_VEL
LIN {X 0,Y 737.349,Z 856.305,A -85,B 0,C 180,E1 1932.248,E2 1932.248} C_VEL
LIN {X 0,Y 735.101,Z 775.388,A -85,B 0,C 180,E1 1933.64,E2 1933.64} C_VEL
LIN {X 0,Y 731.66,Z 767.06,A -85,B 0,C 180,E1 1933.976,E2 1933.976} C_VEL
LIN {X 0,Y 730.831,Z 767.06,A -85,B 0,C 180,E1 1943.72,E2 1943.72} C_VEL
LIN {X 0,Y 730.619,Z 767.06,A -85,B 0,C 180,E1 1952.138,E2 1952.138} C_VEL
LIN {X 0,Y 730.979,Z 767.06,A -85,B 0,C 180,E1 1958.694,E2 1958.694} C_VEL
LIN {X 0,Y 731.383,Z 767.06,A -85,B 0,C 180,E1 1967.41,E2 1967.41} C_VEL
LIN {X 0,Y 731.699,Z 767.06,A -85,B 0,C 180,E1 1977.017,E2 1977.017} C_VEL
LIN {X 0,Y 731.233,Z 767.06,A -85,B 0,C 180,E1 1985.344,E2 1985.344} C_VEL
LIN {X 0,Y 730.258,Z 767.06,A -85,B 0,C 180,E1 1987.364,E2 1987.364} C_VEL
LIN {X 0,Y 722.42,Z 767.06,A -85,B 0,C 180,E1 1990.097,E2 1990.097} C_VEL
LIN {X 0,Y 722.217,Z 767.06,A -85,B 0,C 180,E1 1995.208,E2 1995.208} C_VEL
LIN {X 0,Y 722.689,Z 767.06,A -85,B 0,C 180,E1 2001.537,E2 2001.537} C_VEL
LIN {X 0,Y 722.853,Z 767.06,A -85,B 0,C 180,E1 2009.533,E2 2009.533} C_VEL
LIN {X 0,Y 722.425,Z 767.06,A -85,B 0,C 180,E1 2018.257,E2 2018.257} C_VEL
LIN {X 0,Y 722.667,Z 767.06,A -85,B 0,C 180,E1 2026.38,E2 2026.38} C_VEL
LIN {X 0,Y 722.565,Z 768.848,A -85,B 0,C 180,E1 2031.338,E2 2031.338} C_VEL
LIN {X 0,Y 730.988,Z 786.501,A -85,B 0,C 180,E1 2032.08,E2 2032.08} C_VEL
LIN {X 0,Y 730.383,Z 877.861,A -85,B 0,C 180,E1 2033.592,E2 2033.592} C_VEL
LIN {X 0,Y 728.808,Z 955.015,A -85,B 0,C 180,E1 2036.252,E2 2036.252} C_VEL
LIN {X 0,Y 727.069,Z 1024.618,A -85,B 0,C 180,E1 2040.01,E2 2040.01} C_VEL
LIN {X 0,Y 725.461,Z 1086.18,A -85,B 0,C 180,E1 2044.746,E2 2044.746} C_VEL
LIN {X 0,Y 724.411,Z 1137.93,A -85,B 0,C 180,E1 2050.334,E2 2050.334} C_VEL
LIN {X 0,Y 723.594,Z 1176.205,A -85,B 0,C 180,E1 2056.362,E2 2056.362} C_VEL
LIN {X 0,Y 723.429,Z 1199.02,A -85,B 0,C 180,E1 2062.167,E2 2062.167} C_VEL
LIN {X 0,Y 723.153,Z 1209.402,A -85,B 0,C 180,E1 2068.196,E2 2068.196} C_VEL
LIN {X 0,Y 723.29,Z 1206.834,A -85,B 0,C 180,E1 2074.206,E2 2074.206} C_VEL
LIN {X 0,Y 723.21,Z 1191.083,A -85,B 0,C 180,E1 2080.265,E2 2080.265} C_VEL
LIN {X 0,Y 723.493,Z 1161.77,A -85,B 0,C 180,E1 2086.239,E2 2086.239} C_VEL
LIN {X 0,Y 724.315,Z 1118.898,A -85,B 0,C 180,E1 2091.975,E2 2091.975} C_VEL
LIN {X 0,Y 725.709,Z 1063.146,A -85,B 0,C 180,E1 2097.225,E2 2097.225} C_VEL
LIN {X 0,Y 727.76,Z 996.684,A -85,B 0,C 180,E1 2101.667,E2 2101.667} C_VEL
LIN {X 0,Y 729.665,Z 925.685,A -85,B 0,C 180,E1 2104.912,E2 2104.912} C_VEL
LIN {X 0,Y 731.044,Z 851.926,A -85,B 0,C 180,E1 2106.972,E2 2106.972} C_VEL
LIN {X 0,Y 729.29,Z 780.177,A -85,B 0,C 180,E1 2108.102,E2 2108.102} C_VEL
LIN {X 0,Y 722.914,Z 767.06,A -85,B 0,C 180,E1 2108.817,E2 2108.817} C_VEL
LIN {X 0,Y 722.093,Z 767.06,A -85,B 0,C 180,E1 2115.291,E2 2115.291} C_VEL
LIN {X 0,Y 722.87,Z 767.06,A -85,B 0,C 180,E1 2121.874,E2 2121.874} C_VEL
LIN {X 0,Y 722.559,Z 767.06,A -85,B 0,C 180,E1 2129.062,E2 2129.062} C_VEL
LIN {X 0,Y 722.334,Z 767.06,A -85,B 0,C 180,E1 2135.952,E2 2135.952} C_VEL
LIN {X 0,Y 722.609,Z 767.06,A -85,B 0,C 180,E1 2143.55,E2 2143.55} C_VEL
LIN {X 0,Y 722.837,Z 767.06,A -85,B 0,C 180,E1 2150.957,E2 2150.957} C_VEL
LIN {X 0,Y 723.037,Z 767.06,A -85,B 0,C 180,E1 2158.209,E2 2158.209} C_VEL
LIN {X 0,Y 723.264,Z 767.06,A -85,B 0,C 180,E1 2165.427,E2 2165.427} C_VEL
LIN {X 0,Y 722.63,Z 767.06,A -85,B 0,C 180,E1 2173.981,E2 2173.981} C_VEL
LIN {X 0,Y 722.653,Z 767.06,A -85,B 0,C 180,E1 2181.564,E2 2181.564} C_VEL
LIN {X 0,Y 722.799,Z 767.06,A -85,B 0,C 180,E1 2189.563,E2 2189.563} C_VEL
LIN {X 0,Y 722.475,Z 767.06,A -85,B 0,C 180,E1 2198.285,E2 2198.285} C_VEL
LIN {X 0,Y 722.678,Z 767.06,A -85,B 0,C 180,E1 2206.414,E2 2206.414} C_VEL
LIN {X 0,Y 722.71,Z 767.06,A -85,B 0,C 180,E1 2214.76,E2 2214.76} C_VEL
LIN {X 0,Y 722.902,Z 768.634,A -85,B 0,C 180,E1 2217.436,E2 2217.436} C_VEL
LIN {X 0,Y 730.366,Z 786.858,A -85,B 0,C 180,E1 2218.123,E2 2218.123} C_VEL
LIN {X 0,Y 730.301,Z 873.541,A -85,B 0,C 180,E1 2219.696,E2 2219.696} C_VEL
LIN {X 0,Y 728.743,Z 949.26,A -85,B 0,C 180,E1 2222.404,E2 2222.404} C_VEL
LIN {X 0,Y 726.779,Z 1019.024,A -85,B 0,C 180,E1 2226.253,E2 2226.253} C_VEL
LIN {X 0,Y 725.05,Z 1080.46,A -85,B 0,C 180,E1 2231.086,E2 2231.086} C_VEL
LIN {X 0,Y 723.775,Z 1129.87,A -85,B 0,C 180,E1 2236.523,E2 2236.523} C_VEL
LIN {X 0,Y 723.328,Z 1163.966,A -85,B 0,C 180,E1 2241.866,E2 2241.866} C_VEL
LIN {X 0,Y 723.042,Z 1187.5,A -85,B 0,C 180,E1 2247.598,E2 2247.598} C_VEL
LIN {X 0,Y 723.262,Z 1198.432,A -85,B 0,C 180,E1 2253.006,E2 2253.006} C_VEL
LIN {X 0,Y 723.223,Z 1198.287,A -85,B 0,C 180,E1 2259.05,E2 2259.05} C_VEL
LIN {X 0,Y 723.154,Z 1184.688,A -85,B 0,C 180,E1 2265.198,E2 2265.198} C_VEL
LIN {X 0,Y 723.38,Z 1158.516,A -85,B 0,C 180,E1 2271.04,E2 2271.04} C_VEL
LIN {X 0,Y 724.038,Z 1118.913,A -85,B 0,C 180,E1 2276.765,E2 2276.765} C_VEL
LIN {X 0,Y 725.504,Z 1064.867,A -85,B 0,C 180,E1 2282.211,E2 2282.211} C_VEL
LIN {X 0,Y 727.373,Z 1001.086,A -85,B 0,C 180,E1 2286.789,E2 2286.789} C_VEL
LIN {X 0,Y 729.283,Z 931.793,A -85,B 0,C 180,E1 2290.247,E2 2290.247} C_VEL
LIN {X 0,Y 730.816,Z 858.097,A -85,B 0,C 180,E1 2292.582,E2 2292.582} C_VEL
LIN {X 0,Y 728.725,Z 777.943,A -85,B 0,C 180,E1 2293.997,E2 2293.997} C_VEL
LIN {X 0,Y 723.423,Z 767.06,A -85,B 0,C 180,E1 2294.609,E2 2294.609} C_VEL
LIN {X 0,Y 722.753,Z 767.06,A -85,B 0,C 180,E1 2303.884,E2 2303.884} C_VEL
LIN {X 0,Y 722.756,Z 767.06,A -85,B 0,C 180,E1 2311.808,E2 2311.808} C_VEL
LIN {X 0,Y 722.569,Z 767.06,A -85,B 0,C 180,E1 2319.721,E2 2319.721} C_VEL
LIN {X 0,Y 723.374,Z 767.06,A -85,B 0,C 180,E1 2327.268,E2 2327.268} C_VEL
LIN {X 0,Y 723.658,Z 767.06,A -85,B 0,C 180,E1 2336.984,E2 2336.984} C_VEL
LIN {X 0,Y 723.195,Z 767.06,A -85,B 0,C 180,E1 2345.404,E2 2345.404} C_VEL
LIN {X 0,Y 722.42,Z 767.06,A -85,B 0,C 180,E1 2350.097,E2 2350.097} C_VEL
LIN {X 0,Y 715.188,Z 767.06,A -85,B 0,C 180,E1 2352.875,E2 2352.875} C_VEL
LIN {X 0,Y 714.539,Z 767.06,A -85,B 0,C 180,E1 2361.795,E2 2361.795} C_VEL
LIN {X 0,Y 714.653,Z 767.06,A -85,B 0,C 180,E1 2369.906,E2 2369.906} C_VEL
LIN {X 0,Y 714.689,Z 767.06,A -85,B 0,C 180,E1 2377.277,E2 2377.277} C_VEL
LIN {X 0,Y 714.654,Z 767.06,A -85,B 0,C 180,E1 2386.397,E2 2386.397} C_VEL
LIN {X 0,Y 714.27,Z 768.413,A -85,B 0,C 180,E1 2390.798,E2 2390.798} C_VEL
LIN {X 0,Y 724.692,Z 789.624,A -85,B 0,C 180,E1 2391.729,E2 2391.729} C_VEL
LIN {X 0,Y 723.865,Z 879.025,A -85,B 0,C 180,E1 2393.242,E2 2393.242} C_VEL
LIN {X 0,Y 721.949,Z 955.531,A -85,B 0,C 180,E1 2395.912,E2 2395.912} C_VEL
LIN {X 0,Y 719.826,Z 1024.886,A -85,B 0,C 180,E1 2399.695,E2 2399.695} C_VEL
LIN {X 0,Y 717.872,Z 1086.011,A -85,B 0,C 180,E1 2404.443,E2 2404.443} C_VEL
LIN {X 0,Y 716.71,Z 1137.283,A -85,B 0,C 180,E1 2410.028,E2 2410.028} C_VEL
LIN {X 0,Y 715.714,Z 1176.205,A -85,B 0,C 180,E1 2416.208,E2 2416.208} C_VEL
LIN {X 0,Y 715.458,Z 1199.02,A -85,B 0,C 180,E1 2422.079,E2 2422.079} C_VEL
LIN {X 0,Y 715.173,Z 1209.402,A -85,B 0,C 180,E1 2428.176,E2 2428.176} C_VEL
LIN {X 0,Y 715.276,Z 1206.834,A -85,B 0,C 180,E1 2434.254,E2 2434.254} C_VEL
LIN {X 0,Y 715.196,Z 1191.083,A -85,B 0,C 180,E1 2440.381,E2 2440.381} C_VEL
LIN {X 0,Y 715.538,Z 1161.616,A -85,B 0,C 180,E1 2446.449,E2 2446.449} C_VEL
LIN {X 0,Y 716.535,Z 1119.039,A -85,B 0,C 180,E1 2452.211,E2 2452.211} C_VEL
LIN {X 0,Y 718.227,Z 1063.146,A -85,B 0,C 180,E1 2457.532,E2 2457.532} C_VEL
LIN {X 0,Y 720.7,Z 996.563,A -85,B 0,C 180,E1 2462.021,E2 2462.021} C_VEL
LIN {X 0,Y 722.997,Z 924.688,A -85,B 0,C 180,E1 2465.32,E2 2465.32} C_VEL
LIN {X 0,Y 724.641,Z 851.926,A -85,B 0,C 180,E1 2467.354,E2 2467.354} C_VEL
LIN {X 0,Y 723.169,Z 783.427,A -85,B 0,C 180,E1 2468.443,E2 2468.443} C_VEL
LIN {X 0,Y 714.9,Z 767.06,A -85,B 0,C 180,E1 2469.264,E2 2469.264} C_VEL
LIN {X 0,Y 714.013,Z 767.06,A -85,B 0,C 180,E1 2476.352,E2 2476.352} C_VEL
LIN {X 0,Y 714.659,Z 767.06,A -85,B 0,C 180,E1 2482.793,E2 2482.793} C_VEL
LIN {X 0,Y 714.44,Z 767.06,A -85,B 0,C 180,E1 2490.084,E2 2490.084} C_VEL
LIN {X 0,Y 714.043,Z 767.06,A -85,B 0,C 180,E1 2496.872,E2 2496.872} C_VEL
LIN {X 0,Y 714.699,Z 767.06,A -85,B 0,C 180,E1 2503.363,E2 2503.363} C_VEL
LIN {X 0,Y 714.859,Z 767.06,A -85,B 0,C 180,E1 2510.855,E2 2510.855} C_VEL
LIN {X 0,Y 715.04,Z 767.06,A -85,B 0,C 180,E1 2518.189,E2 2518.189} C_VEL
LIN {X 0,Y 715.212,Z 767.06,A -85,B 0,C 180,E1 2525.489,E2 2525.489} C_VEL
LIN {X 0,Y 715.228,Z 767.06,A -85,B 0,C 180,E1 2532.879,E2 2532.879} C_VEL
LIN {X 0,Y 714.507,Z 767.06,A -85,B 0,C 180,E1 2541.822,E2 2541.822} C_VEL
LIN {X 0,Y 714.582,Z 767.06,A -85,B 0,C 180,E1 2549.937,E2 2549.937} C_VEL
LIN {X 0,Y 714.722,Z 767.06,A -85,B 0,C 180,E1 2557.286,E2 2557.286} C_VEL
LIN {X 0,Y 714.682,Z 767.06,A -85,B 0,C 180,E1 2566.404,E2 2566.404} C_VEL
LIN {X 0,Y 714.697,Z 767.06,A -85,B 0,C 180,E1 2574.818,E2 2574.818} C_VEL
LIN {X 0,Y 714.8,Z 768.808,A -85,B 0,C 180,E1 2576.919,E2 2576.919} C_VEL
LIN {X 0,Y 724.067,Z 788.248,A -85,B 0,C 180,E1 2577.752,E2 2577.752} C_VEL
LIN {X 0,Y 723.735,Z 874.386,A -85,B 0,C 180,E1 2579.338,E2 2579.338} C_VEL
LIN {X 0,Y 721.81,Z 950.876,A -85,B 0,C 180,E1 2582.116,E2 2582.116} C_VEL
LIN {X 0,Y 719.487,Z 1020.225,A -85,B 0,C 180,E1 2586.004,E2 2586.004} C_VEL
LIN {X 0,Y 717.44,Z 1081.24,A -85,B 0,C 180,E1 2590.877,E2 2590.877} C_VEL
LIN {X 0,Y 715.946,Z 1130.408,A -85,B 0,C 180,E1 2596.372,E2 2596.372} C_VEL
LIN {X 0,Y 715.39,Z 1164.309,A -85,B 0,C 180,E1 2601.775,E2 2601.775} C_VEL
LIN {X 0,Y 715.06,Z 1187.702,A -85,B 0,C 180,E1 2607.571,E2 2607.571} C_VEL
LIN {X 0,Y 715.252,Z 1198.498,A -85,B 0,C 180,E1 2613.04,E2 2613.04} C_VEL
LIN {X 0,Y 715.069,Z 1197.933,A -85,B 0,C 180,E1 2619.389,E2 2619.389} C_VEL
LIN {X 0,Y 715.074,Z 1184.455,A -85,B 0,C 180,E1 2625.374,E2 2625.374} C_VEL
LIN {X 0,Y 715.447,Z 1159.247,A -85,B 0,C 180,E1 2631.081,E2 2631.081} C_VEL
LIN {X 0,Y 716.247,Z 1120.998,A -85,B 0,C 180,E1 2636.75,E2 2636.75} C_VEL
LIN {X 0,Y 717.86,Z 1068.154,A -85,B 0,C 180,E1 2642.224,E2 2642.224} C_VEL
LIN {X 0,Y 720.124,Z 1003.494,A -85,B 0,C 180,E1 2646.98,E2 2646.98} C_VEL
LIN {X 0,Y 722.466,Z 933.183,A -85,B 0,C 180,E1 2650.557,E2 2650.557} C_VEL
LIN {X 0,Y 724.345,Z 858.588,A -85,B 0,C 180,E1 2652.951,E2 2652.951} C_VEL
LIN {X 0,Y 722.769,Z 781.937,A -85,B 0,C 180,E1 2654.317,E2 2654.317} C_VEL
LIN {X 0,Y 715.286,Z 767.06,A -85,B 0,C 180,E1 2655.015,E2 2655.015} C_VEL
LIN {X 0,Y 714.626,Z 767.06,A -85,B 0,C 180,E1 2664.273,E2 2664.273} C_VEL
LIN {X 0,Y 714.766,Z 767.06,A -85,B 0,C 180,E1 2671.703,E2 2671.703} C_VEL
LIN {X 0,Y 714.657,Z 767.06,A -85,B 0,C 180,E1 2679.487,E2 2679.487} C_VEL
LIN {X 0,Y 715.411,Z 767.06,A -85,B 0,C 180,E1 2687.124,E2 2687.124} C_VEL
LIN {X 0,Y 715.617,Z 767.06,A -85,B 0,C 180,E1 2696.95,E2 2696.95} C_VEL
LIN {X 0,Y 715.143,Z 767.06,A -85,B 0,C 180,E1 2705.465,E2 2705.465} C_VEL
LIN {X 0,Y 715.188,Z 767.06,A -85,B 0,C 180,E1 2712.875,E2 2712.875} C_VEL
LIN {X 0,Y 706.141,Z 767.06,A -85,B 0,C 180,E1 2715.638,E2 2715.638} C_VEL
LIN {X 0,Y 706.42,Z 767.06,A -85,B 0,C 180,E1 2722.059,E2 2722.059} C_VEL
LIN {X 0,Y 706.484,Z 767.06,A -85,B 0,C 180,E1 2730.288,E2 2730.288} C_VEL
LIN {X 0,Y 706.269,Z 767.06,A -85,B 0,C 180,E1 2738.396,E2 2738.396} C_VEL
LIN {X 0,Y 706.72,Z 767.06,A -85,B 0,C 180,E1 2745.956,E2 2745.956} C_VEL
LIN {X 0,Y 706.23,Z 768.907,A -85,B 0,C 180,E1 2750.27,E2 2750.27} C_VEL
LIN {X 0,Y 718.444,Z 793.745,A -85,B 0,C 180,E1 2751.387,E2 2751.387} C_VEL
LIN {X 0,Y 717.318,Z 880.804,A -85,B 0,C 180,E1 2752.9,E2 2752.9} C_VEL
LIN {X 0,Y 715.026,Z 957.836,A -85,B 0,C 180,E1 2755.647,E2 2755.647} C_VEL
LIN {X 0,Y 712.503,Z 1027.622,A -85,B 0,C 180,E1 2759.542,E2 2759.542} C_VEL
LIN {X 0,Y 710.231,Z 1088.333,A -85,B 0,C 180,E1 2764.371,E2 2764.371} C_VEL
LIN {X 0,Y 708.746,Z 1139.954,A -85,B 0,C 180,E1 2770.15,E2 2770.15} C_VEL
LIN {X 0,Y 707.636,Z 1177.763,A -85,B 0,C 180,E1 2776.364,E2 2776.364} C_VEL
LIN {X 0,Y 707.219,Z 1200.659,A -85,B 0,C 180,E1 2782.606,E2 2782.606} C_VEL
LIN {X 0,Y 707.177,Z 1209.402,A -85,B 0,C 180,E1 2788.155,E2 2788.155} C_VEL
LIN {X 0,Y 707.238,Z 1206.739,A -85,B 0,C 180,E1 2794.364,E2 2794.364} C_VEL
LIN {X 0,Y 707.157,Z 1191.082,A -85,B 0,C 180,E1 2800.501,E2 2800.501} C_VEL
LIN {X 0,Y 707.605,Z 1162.497,A -85,B 0,C 180,E1 2806.495,E2 2806.495} C_VEL
LIN {X 0,Y 708.764,Z 1120.701,A -85,B 0,C 180,E1 2812.279,E2 2812.279} C_VEL
LIN {X 0,Y 710.715,Z 1065.122,A -85,B 0,C 180,E1 2817.686,E2 2817.686} C_VEL
LIN {X 0,Y 713.57,Z 998.365,A -85,B 0,C 180,E1 2822.273,E2 2822.273} C_VEL
LIN {X 0,Y 716.292,Z 925.949,A -85,B 0,C 180,E1 2825.652,E2 2825.652} C_VEL
LIN {X 0,Y 718.204,Z 853.648,A -85,B 0,C 180,E1 2827.712,E2 2827.712} C_VEL
LIN {X 0,Y 716.864,Z 786.83,A -85,B 0,C 180,E1 2828.801,E2 2828.801} C_VEL
LIN {X 0,Y 706.904,Z 767.06,A -85,B 0,C 180,E1 2829.873,E2 2829.873} C_VEL
LIN {X 0,Y 706.265,Z 767.06,A -85,B 0,C 180,E1 2837.794,E2 2837.794} C_VEL
LIN {X 0,Y 706.975,Z 767.06,A -85,B 0,C 180,E1 2845.669,E2 2845.669} C_VEL
LIN {X 0,Y 706.888,Z 767.06,A -85,B 0,C 180,E1 2853.917,E2 2853.917} C_VEL
LIN {X 0,Y 706.744,Z 767.06,A -85,B 0,C 180,E1 2863.17,E2 2863.17} C_VEL
LIN {X 0,Y 706.893,Z 767.06,A -85,B 0,C 180,E1 2870.751,E2 2870.751} C_VEL
LIN {X 0,Y 707.044,Z 767.06,A -85,B 0,C 180,E1 2878.168,E2 2878.168} C_VEL
LIN {X 0,Y 707.184,Z 767.06,A -85,B 0,C 180,E1 2885.551,E2 2885.551} C_VEL
LIN {X 0,Y 707.146,Z 767.06,A -85,B 0,C 180,E1 2893.029,E2 2893.029} C_VEL
LIN {X 0,Y 706.765,Z 767.06,A -85,B 0,C 180,E1 2901.042,E2 2901.042} C_VEL
LIN {X 0,Y 706.635,Z 767.06,A -85,B 0,C 180,E1 2909.645,E2 2909.645} C_VEL
LIN {X 0,Y 706.317,Z 767.06,A -85,B 0,C 180,E1 2918.407,E2 2918.407} C_VEL
LIN {X 0,Y 706.768,Z 767.06,A -85,B 0,C 180,E1 2925.987,E2 2925.987} C_VEL
LIN {X 0,Y 706.793,Z 767.06,A -85,B 0,C 180,E1 2933.843,E2 2933.843} C_VEL
LIN {X 0,Y 706.703,Z 768.508,A -85,B 0,C 180,E1 2936.381,E2 2936.381} C_VEL
LIN {X 0,Y 717.834,Z 792.037,A -85,B 0,C 180,E1 2937.407,E2 2937.407} C_VEL
LIN {X 0,Y 717.183,Z 876.48,A -85,B 0,C 180,E1 2939.01,E2 2939.01} C_VEL
LIN {X 0,Y 714.903,Z 951.744,A -85,B 0,C 180,E1 2941.786,E2 2941.786} C_VEL
LIN {X 0,Y 712.157,Z 1022.215,A -85,B 0,C 180,E1 2945.804,E2 2945.804} C_VEL
LIN {X 0,Y 709.747,Z 1083.711,A -85,B 0,C 180,E1 2950.824,E2 2950.824} C_VEL
LIN {X 0,Y 708.073,Z 1132.126,A -85,B 0,C 180,E1 2956.376,E2 2956.376} C_VEL
LIN {X 0,Y 707.29,Z 1166.184,A -85,B 0,C 180,E1 2961.991,E2 2961.991} C_VEL
LIN {X 0,Y 707.084,Z 1187.903,A -85,B 0,C 180,E1 2967.543,E2 2967.543} C_VEL
LIN {X 0,Y 706.944,Z 1199.101,A -85,B 0,C 180,E1 2973.675,E2 2973.675} C_VEL
LIN {X 0,Y 707.128,Z 1198.146,A -85,B 0,C 180,E1 2979.257,E2 2979.257} C_VEL
LIN {X 0,Y 707.147,Z 1185.211,A -85,B 0,C 180,E1 2985.249,E2 2985.249} C_VEL
LIN {X 0,Y 707.505,Z 1160.004,A -85,B 0,C 180,E1 2991.119,E2 2991.119} C_VEL
LIN {X 0,Y 708.421,Z 1121.215,A -85,B 0,C 180,E1 2996.964,E2 2996.964} C_VEL
LIN {X 0,Y 710.38,Z 1067.669,A -85,B 0,C 180,E1 3002.565,E2 3002.565} C_VEL
LIN {X 0,Y 712.98,Z 1003.655,A -85,B 0,C 180,E1 3007.316,E2 3007.316} C_VEL
LIN {X 0,Y 715.666,Z 934.384,A -85,B 0,C 180,E1 3010.881,E2 3010.881} C_VEL
LIN {X 0,Y 717.864,Z 860.171,A -85,B 0,C 180,E1 3013.303,E2 3013.303} C_VEL
LIN {X 0,Y 716.553,Z 785.207,A -85,B 0,C 180,E1 3014.671,E2 3014.671} C_VEL
LIN {X 0,Y 707.031,Z 767.06,A -85,B 0,C 180,E1 3015.631,E2 3015.631} C_VEL
LIN {X 0,Y 706.656,Z 767.06,A -85,B 0,C 180,E1 3023.807,E2 3023.807} C_VEL
LIN {X 0,Y 706.794,Z 767.06,A -85,B 0,C 180,E1 3031.113,E2 3031.113} C_VEL
LIN {X 0,Y 706.691,Z 767.06,A -85,B 0,C 180,E1 3039.245,E2 3039.245} C_VEL
LIN {X 0,Y 707.4,Z 767.06,A -85,B 0,C 180,E1 3047.269,E2 3047.269} C_VEL
LIN {X 0,Y 707.573,Z 767.06,A -85,B 0,C 180,E1 3056.923,E2 3056.923} C_VEL
LIN {X 0,Y 707.105,Z 767.06,A -85,B 0,C 180,E1 3065.527,E2 3065.527} C_VEL
LIN {X 0,Y 707.121,Z 767.06,A -85,B 0,C 180,E1 3073.004,E2 3073.004} C_VEL
LIN {X 0,Y 706.141,Z 767.06,A -85,B 0,C 180,E1 3075.638,E2 3075.638} C_VEL
LIN {X 0,Y 698.546,Z 767.06,A -85,B 0,C 180,E1 3078.462,E2 3078.462} C_VEL
LIN {X 0,Y 698.378,Z 767.06,A -85,B 0,C 180,E1 3086.426,E2 3086.426} C_VEL
LIN {X 0,Y 698.124,Z 767.06,A -85,B 0,C 180,E1 3093.631,E2 3093.631} C_VEL
LIN {X 0,Y 697.857,Z 767.06,A -85,B 0,C 180,E1 3099.866,E2 3099.866} C_VEL
LIN {X 0,Y 698.388,Z 767.06,A -85,B 0,C 180,E1 3106.842,E2 3106.842} C_VEL
LIN {X 0,Y 698.153,Z 768.858,A -85,B 0,C 180,E1 3109.716,E2 3109.716} C_VEL
LIN {X 0,Y 712.209,Z 795.026,A -85,B 0,C 180,E1 3111.001,E2 3111.001} C_VEL
LIN {X 0,Y 710.896,Z 880.802,A -85,B 0,C 180,E1 3112.508,E2 3112.508} C_VEL
LIN {X 0,Y 708.293,Z 957.183,A -85,B 0,C 180,E1 3115.243,E2 3115.243} C_VEL
LIN {X 0,Y 705.384,Z 1025.886,A -85,B 0,C 180,E1 3119.078,E2 3119.078} C_VEL
LIN {X 0,Y 702.713,Z 1086.658,A -85,B 0,C 180,E1 3123.914,E2 3123.914} C_VEL
LIN {X 0,Y 701.032,Z 1137.454,A -85,B 0,C 180,E1 3129.584,E2 3129.584} C_VEL
LIN {X 0,Y 699.937,Z 1176.208,A -85,B 0,C 180,E1 3135.891,E2 3135.891} C_VEL
LIN {X 0,Y 699.516,Z 1199.021,A -85,B 0,C 180,E1 3141.898,E2 3141.898} C_VEL
LIN {X 0,Y 699.197,Z 1209.402,A -85,B 0,C 180,E1 3148.134,E2 3148.134} C_VEL
LIN {X 0,Y 699.265,Z 1206.834,A -85,B 0,C 180,E1 3154.351,E2 3154.351} C_VEL
LIN {X 0,Y 699.166,Z 1191.082,A -85,B 0,C 180,E1 3160.622,E2 3160.622} C_VEL
LIN {X 0,Y 699.655,Z 1162.495,A -85,B 0,C 180,E1 3166.688,E2 3166.688} C_VEL
LIN {X 0,Y 700.997,Z 1121.216,A -85,B 0,C 180,E1 3172.48,E2 3172.48} C_VEL
LIN {X 0,Y 703.279,Z 1066.285,A -85,B 0,C 180,E1 3177.907,E2 3177.907} C_VEL
LIN {X 0,Y 706.454,Z 1001.133,A -85,B 0,C 180,E1 3182.473,E2 3182.473} C_VEL
LIN {X 0,Y 709.512,Z 930.236,A -85,B 0,C 180,E1 3185.878,E2 3185.878} C_VEL
LIN {X 0,Y 711.807,Z 855.626,A -85,B 0,C 180,E1 3188.069,E2 3188.069} C_VEL
LIN {X 0,Y 710.703,Z 790.145,A -85,B 0,C 180,E1 3189.159,E2 3189.159} C_VEL
LIN {X 0,Y 698.975,Z 767.06,A -85,B 0,C 180,E1 3190.436,E2 3190.436} C_VEL
LIN {X 0,Y 698.902,Z 767.06,A -85,B 0,C 180,E1 3200.375,E2 3200.375} C_VEL
LIN {X 0,Y 698.782,Z 767.06,A -85,B 0,C 180,E1 3207.886,E2 3207.886} C_VEL
LIN {X 0,Y 698.589,Z 767.06,A -85,B 0,C 180,E1 3214.964,E2 3214.964} C_VEL
LIN {X 0,Y 698.819,Z 767.06,A -85,B 0,C 180,E1 3222.973,E2 3222.973} C_VEL
LIN {X 0,Y 698.869,Z 767.06,A -85,B 0,C 180,E1 3230.845,E2 3230.845} C_VEL
LIN {X 0,Y 699.067,Z 767.06,A -85,B 0,C 180,E1 3238.147,E2 3238.147} C_VEL
LIN {X 0,Y 699.132,Z 767.06,A -85,B 0,C 180,E1 3245.615,E2 3245.615} C_VEL
LIN {X 0,Y 699.042,Z 767.06,A -85,B 0,C 180,E1 3253.183,E2 3253.183} C_VEL
LIN {X 0,Y 698.806,Z 767.06,A -85,B 0,C 180,E1 3261,E2 3261} C_VEL
LIN {X 0,Y 698.734,Z 767.06,A -85,B 0,C 180,E1 3269.253,E2 3269.253} C_VEL
LIN {X 0,Y 698.356,Z 767.06,A -85,B 0,C 180,E1 3278.261,E2 3278.261} C_VEL
LIN {X 0,Y 698.477,Z 767.06,A -85,B 0,C 180,E1 3286.854,E2 3286.854} C_VEL
LIN {X 0,Y 698.612,Z 767.06,A -85,B 0,C 180,E1 3294.887,E2 3294.887} C_VEL
LIN {X 0,Y 698.764,Z 768.757,A -85,B 0,C 180,E1 3295.844,E2 3295.844} C_VEL
LIN {X 0,Y 711.654,Z 795.073,A -85,B 0,C 180,E1 3297.048,E2 3297.048} C_VEL
LIN {X 0,Y 710.671,Z 878.379,A -85,B 0,C 180,E1 3298.67,E2 3298.67} C_VEL
LIN {X 0,Y 708.007,Z 953.998,A -85,B 0,C 180,E1 3301.518,E2 3301.518} C_VEL
LIN {X 0,Y 704.85,Z 1024.256,A -85,B 0,C 180,E1 3305.603,E2 3305.603} C_VEL
LIN {X 0,Y 702.171,Z 1084.478,A -85,B 0,C 180,E1 3310.609,E2 3310.609} C_VEL
LIN {X 0,Y 700.19,Z 1133.82,A -85,B 0,C 180,E1 3316.379,E2 3316.379} C_VEL
LIN {X 0,Y 699.236,Z 1168.058,A -85,B 0,C 180,E1 3322.212,E2 3322.212} C_VEL
LIN {X 0,Y 699.111,Z 1188.105,A -85,B 0,C 180,E1 3327.515,E2 3327.515} C_VEL
LIN {X 0,Y 699.206,Z 1198.629,A -85,B 0,C 180,E1 3333.11,E2 3333.11} C_VEL
LIN {X 0,Y 699.077,Z 1198.06,A -85,B 0,C 180,E1 3339.365,E2 3339.365} C_VEL
LIN {X 0,Y 699.111,Z 1185.176,A -85,B 0,C 180,E1 3345.368,E2 3345.368} C_VEL
LIN {X 0,Y 699.551,Z 1160.716,A -85,B 0,C 180,E1 3351.165,E2 3351.165} C_VEL
LIN {X 0,Y 700.61,Z 1122.287,A -85,B 0,C 180,E1 3357.074,E2 3357.074} C_VEL
LIN {X 0,Y 702.837,Z 1069.141,A -85,B 0,C 180,E1 3362.741,E2 3362.741} C_VEL
LIN {X 0,Y 705.802,Z 1004.895,A -85,B 0,C 180,E1 3367.59,E2 3367.59} C_VEL
LIN {X 0,Y 708.915,Z 934.67,A -85,B 0,C 180,E1 3371.25,E2 3371.25} C_VEL
LIN {X 0,Y 711.455,Z 859.888,A -85,B 0,C 180,E1 3373.704,E2 3373.704} C_VEL
LIN {X 0,Y 710.449,Z 788.384,A -85,B 0,C 180,E1 3375.026,E2 3375.026} C_VEL
LIN {X 0,Y 698.781,Z 767.06,A -85,B 0,C 180,E1 3376.19,E2 3376.19} C_VEL
LIN {X 0,Y 698.393,Z 767.06,A -85,B 0,C 180,E1 3384.846,E2 3384.846} C_VEL
LIN {X 0,Y 698.515,Z 767.06,A -85,B 0,C 180,E1 3392.154,E2 3392.154} C_VEL
LIN {X 0,Y 698.75,Z 767.06,A -85,B 0,C 180,E1 3398.998,E2 3398.998} C_VEL
LIN {X 0,Y 699.434,Z 767.06,A -85,B 0,C 180,E1 3408.098,E2 3408.098} C_VEL
LIN {X 0,Y 699.125,Z 767.06,A -85,B 0,C 180,E1 3418.123,E2 3418.123} C_VEL
LIN {X 0,Y 699.054,Z 767.06,A -85,B 0,C 180,E1 3425.591,E2 3425.591} C_VEL
LIN {X 0,Y 699.018,Z 767.06,A -85,B 0,C 180,E1 3433.158,E2 3433.158} C_VEL
LIN {X 0,Y 698.546,Z 767.06,A -85,B 0,C 180,E1 3438.462,E2 3438.462} C_VEL
LIN {X 0,Y 690.67,Z 767.06,A -85,B 0,C 180,E1 3441.323,E2 3441.323} C_VEL
LIN {X 0,Y 690.566,Z 767.06,A -85,B 0,C 180,E1 3449.838,E2 3449.838} C_VEL
LIN {X 0,Y 690.548,Z 767.06,A -85,B 0,C 180,E1 3457.146,E2 3457.146} C_VEL
LIN {X 0,Y 690.464,Z 767.06,A -85,B 0,C 180,E1 3466.222,E2 3466.222} C_VEL
LIN {X 0,Y 690.201,Z 769.06,A -85,B 0,C 180,E1 3469.157,E2 3469.157} C_VEL
LIN {X 0,Y 705.995,Z 799.412,A -85,B 0,C 180,E1 3470.648,E2 3470.648} C_VEL
LIN {X 0,Y 704.285,Z 884.23,A -85,B 0,C 180,E1 3472.195,E2 3472.195} C_VEL
LIN {X 0,Y 701.308,Z 961.03,A -85,B 0,C 180,E1 3475.037,E2 3475.037} C_VEL
LIN {X 0,Y 697.991,Z 1030.332,A -85,B 0,C 180,E1 3479.034,E2 3479.034} C_VEL
LIN {X 0,Y 694.973,Z 1091.957,A -85,B 0,C 180,E1 3484.123,E2 3484.123} C_VEL
LIN {X 0,Y 693.157,Z 1141.116,A -85,B 0,C 180,E1 3489.842,E2 3489.842} C_VEL
LIN {X 0,Y 691.865,Z 1177.765,A -85,B 0,C 180,E1 3496.047,E2 3496.047} C_VEL
LIN {X 0,Y 691.298,Z 1200.653,A -85,B 0,C 180,E1 3502.435,E2 3502.435} C_VEL
LIN {X 0,Y 691.201,Z 1209.402,A -85,B 0,C 180,E1 3508.112,E2 3508.112} C_VEL
LIN {X 0,Y 691.246,Z 1206.834,A -85,B 0,C 180,E1 3514.402,E2 3514.402} C_VEL
LIN {X 0,Y 691.144,Z 1191.08,A -85,B 0,C 180,E1 3520.747,E2 3520.747} C_VEL
LIN {X 0,Y 691.747,Z 1164.396,A -85,B 0,C 180,E1 3526.556,E2 3526.556} C_VEL
LIN {X 0,Y 693.191,Z 1123.144,A -85,B 0,C 180,E1 3532.508,E2 3532.508} C_VEL
LIN {X 0,Y 695.751,Z 1068.802,A -85,B 0,C 180,E1 3538.024,E2 3538.024} C_VEL
LIN {X 0,Y 699.359,Z 1002.891,A -85,B 0,C 180,E1 3542.737,E2 3542.737} C_VEL
LIN {X 0,Y 702.829,Z 931.992,A -85,B 0,C 180,E1 3546.203,E2 3546.203} C_VEL
LIN {X 0,Y 705.406,Z 857.905,A -85,B 0,C 180,E1 3548.425,E2 3548.425} C_VEL
LIN {X 0,Y 704.407,Z 793.049,A -85,B 0,C 180,E1 3549.54,E2 3549.54} C_VEL
LIN {X 0,Y 691.028,Z 767.06,A -85,B 0,C 180,E1 3550.906,E2 3550.906} C_VEL
LIN {X 0,Y 690.772,Z 767.06,A -85,B 0,C 180,E1 3561.273,E2 3561.273} C_VEL
LIN {X 0,Y 690.561,Z 767.06,A -85,B 0,C 180,E1 3568.938,E2 3568.938} C_VEL
LIN {X 0,Y 690.247,Z 767.06,A -85,B 0,C 180,E1 3576.026,E2 3576.026} C_VEL
LIN {X 0,Y 690.846,Z 767.06,A -85,B 0,C 180,E1 3582.771,E2 3582.771} C_VEL
LIN {X 0,Y 690.919,Z 767.06,A -85,B 0,C 180,E1 3590.535,E2 3590.535} C_VEL
LIN {X 0,Y 691.071,Z 767.06,A -85,B 0,C 180,E1 3598.126,E2 3598.126} C_VEL
LIN {X 0,Y 691.101,Z 767.06,A -85,B 0,C 180,E1 3605.681,E2 3605.681} C_VEL
LIN {X 0,Y 690.944,Z 767.06,A -85,B 0,C 180,E1 3613.34,E2 3613.34} C_VEL
LIN {X 0,Y 690.692,Z 767.06,A -85,B 0,C 180,E1 3621.259,E2 3621.259} C_VEL
LIN {X 0,Y 690.49,Z 767.06,A -85,B 0,C 180,E1 3629.834,E2 3629.834} C_VEL
LIN {X 0,Y 690.591,Z 767.06,A -85,B 0,C 180,E1 3637.175,E2 3637.175} C_VEL
LIN {X 0,Y 690.554,Z 767.06,A -85,B 0,C 180,E1 3646.235,E2 3646.235} C_VEL
LIN {X 0,Y 690.63,Z 767.06,A -85,B 0,C 180,E1 3654.974,E2 3654.974} C_VEL
LIN {X 0,Y 691.526,Z 770.772,A -85,B 0,C 180,E1 3655.364,E2 3655.364} C_VEL
LIN {X 0,Y 705.477,Z 797.743,A -85,B 0,C 180,E1 3656.676,E2 3656.676} C_VEL
LIN {X 0,Y 704.197,Z 880.315,A -85,B 0,C 180,E1 3658.327,E2 3658.327} C_VEL
LIN {X 0,Y 701.131,Z 955.608,A -85,B 0,C 180,E1 3661.212,E2 3661.212} C_VEL
LIN {X 0,Y 697.592,Z 1025.596,A -85,B 0,C 180,E1 3665.35,E2 3665.35} C_VEL
LIN {X 0,Y 694.458,Z 1086.909,A -85,B 0,C 180,E1 3670.55,E2 3670.55} C_VEL
LIN {X 0,Y 692.298,Z 1135.42,A -85,B 0,C 180,E1 3676.382,E2 3676.382} C_VEL
LIN {X 0,Y 691.292,Z 1168.399,A -85,B 0,C 180,E1 3682.122,E2 3682.122} C_VEL
LIN {X 0,Y 691.151,Z 1188.306,A -85,B 0,C 180,E1 3687.487,E2 3687.487} C_VEL
LIN {X 0,Y 691.2,Z 1198.695,A -85,B 0,C 180,E1 3693.146,E2 3693.146} C_VEL
LIN {X 0,Y 691.03,Z 1197.974,A -85,B 0,C 180,E1 3699.475,E2 3699.475} C_VEL
LIN {X 0,Y 691.056,Z 1184.81,A -85,B 0,C 180,E1 3705.594,E2 3705.594} C_VEL
LIN {X 0,Y 691.622,Z 1161.419,A -85,B 0,C 180,E1 3711.212,E2 3711.212} C_VEL
LIN {X 0,Y 692.759,Z 1122.473,A -85,B 0,C 180,E1 3717.301,E2 3717.301} C_VEL
LIN {X 0,Y 695.287,Z 1069.916,A -85,B 0,C 180,E1 3722.984,E2 3722.984} C_VEL
LIN {X 0,Y 698.658,Z 1005.809,A -85,B 0,C 180,E1 3727.891,E2 3727.891} C_VEL
LIN {X 0,Y 702.18,Z 936.054,A -85,B 0,C 180,E1 3731.578,E2 3731.578} C_VEL
LIN {X 0,Y 705.041,Z 862.098,A -85,B 0,C 180,E1 3734.052,E2 3734.052} C_VEL
LIN {X 0,Y 704.257,Z 791.91,A -85,B 0,C 180,E1 3735.39,E2 3735.39} C_VEL
LIN {X 0,Y 690.543,Z 767.06,A -85,B 0,C 180,E1 3736.825,E2 3736.825} C_VEL
LIN {X 0,Y 690.494,Z 767.06,A -85,B 0,C 180,E1 3744.383,E2 3744.383} C_VEL
LIN {X 0,Y 690.585,Z 767.06,A -85,B 0,C 180,E1 3751.806,E2 3751.806} C_VEL
LIN {X 0,Y 690.448,Z 767.06,A -85,B 0,C 180,E1 3760.078,E2 3760.078} C_VEL
LIN {X 0,Y 691.411,Z 767.06,A -85,B 0,C 180,E1 3767.958,E2 3767.958} C_VEL
LIN {X 0,Y 691.129,Z 767.06,A -85,B 0,C 180,E1 3778.101,E2 3778.101} C_VEL
LIN {X 0,Y 691.034,Z 767.06,A -85,B 0,C 180,E1 3785.656,E2 3785.656} C_VEL
LIN {X 0,Y 690.922,Z 767.06,A -85,B 0,C 180,E1 3793.315,E2 3793.315} C_VEL
LIN {X 0,Y 690.67,Z 767.06,A -85,B 0,C 180,E1 3801.323,E2 3801.323} C_VEL
LIN {X 0,Y 681.97,Z 767.06,A -85,B 0,C 180,E1 3804.195,E2 3804.195} C_VEL
LIN {X 0,Y 682.148,Z 767.06,A -85,B 0,C 180,E1 3811.489,E2 3811.489} C_VEL
LIN {X 0,Y 682.289,Z 767.06,A -85,B 0,C 180,E1 3817.903,E2 3817.903} C_VEL
LIN {X 0,Y 682.458,Z 767.06,A -85,B 0,C 180,E1 3826.231,E2 3826.231} C_VEL
LIN {X 0,Y 682.247,Z 769.062,A -85,B 0,C 180,E1 3828.577,E2 3828.577} C_VEL
LIN {X 0,Y 699.846,Z 803.175,A -85,B 0,C 180,E1 3830.284,E2 3830.284} C_VEL
LIN {X 0,Y 697.763,Z 887.213,A -85,B 0,C 180,E1 3831.869,E2 3831.869} C_VEL
LIN {X 0,Y 694.37,Z 964.089,A -85,B 0,C 180,E1 3834.791,E2 3834.791} C_VEL
LIN {X 0,Y 690.581,Z 1033.972,A -85,B 0,C 180,E1 3838.931,E2 3838.931} C_VEL
LIN {X 0,Y 687.305,Z 1094.271,A -85,B 0,C 180,E1 3844.045,E2 3844.045} C_VEL
LIN {X 0,Y 685.158,Z 1143.522,A -85,B 0,C 180,E1 3849.935,E2 3849.935} C_VEL
LIN {X 0,Y 683.804,Z 1179.306,A -85,B 0,C 180,E1 3856.206,E2 3856.206} C_VEL
LIN {X 0,Y 683.336,Z 1200.65,A -85,B 0,C 180,E1 3862.346,E2 3862.346} C_VEL
LIN {X 0,Y 683.208,Z 1209.402,A -85,B 0,C 180,E1 3868.09,E2 3868.09} C_VEL
LIN {X 0,Y 683.216,Z 1206.832,A -85,B 0,C 180,E1 3874.454,E2 3874.454} C_VEL
LIN {X 0,Y 683.231,Z 1192.194,A -85,B 0,C 180,E1 3880.549,E2 3880.549} C_VEL
LIN {X 0,Y 683.838,Z 1164.397,A -85,B 0,C 180,E1 3886.753,E2 3886.753} C_VEL
LIN {X 0,Y 685.391,Z 1124.98,A -85,B 0,C 180,E1 3892.544,E2 3892.544} C_VEL
LIN {X 0,Y 688.157,Z 1071.905,A -85,B 0,C 180,E1 3898.074,E2 3898.074} C_VEL
LIN {X 0,Y 692.146,Z 1007.26,A -85,B 0,C 180,E1 3902.847,E2 3902.847} C_VEL
LIN {X 0,Y 696.054,Z 935.524,A -85,B 0,C 180,E1 3906.463,E2 3906.463} C_VEL
LIN {X 0,Y 698.992,Z 860.628,A -85,B 0,C 180,E1 3908.777,E2 3908.777} C_VEL
LIN {X 0,Y 698.205,Z 796.32,A -85,B 0,C 180,E1 3909.918,E2 3909.918} C_VEL
LIN {X 0,Y 683.002,Z 767.06,A -85,B 0,C 180,E1 3911.451,E2 3911.451} C_VEL
LIN {X 0,Y 682.703,Z 767.06,A -85,B 0,C 180,E1 3920.728,E2 3920.728} C_VEL
LIN {X 0,Y 682.586,Z 767.06,A -85,B 0,C 180,E1 3928.793,E2 3928.793} C_VEL
LIN {X 0,Y 682.365,Z 767.06,A -85,B 0,C 180,E1 3935.731,E2 3935.731} C_VEL
LIN {X 0,Y 682.468,Z 767.06,A -85,B 0,C 180,E1 3943.883,E2 3943.883} C_VEL
LIN {X 0,Y 682.495,Z 767.06,A -85,B 0,C 180,E1 3951.707,E2 3951.707} C_VEL
LIN {X 0,Y 683.079,Z 767.06,A -85,B 0,C 180,E1 3958.104,E2 3958.104} C_VEL
LIN {X 0,Y 683.051,Z 767.06,A -85,B 0,C 180,E1 3965.748,E2 3965.748} C_VEL
LIN {X 0,Y 682.852,Z 767.06,A -85,B 0,C 180,E1 3973.501,E2 3973.501} C_VEL
LIN {X 0,Y 682.559,Z 767.06,A -85,B 0,C 180,E1 3981.525,E2 3981.525} C_VEL
LIN {X 0,Y 682.427,Z 767.06,A -85,B 0,C 180,E1 3990.022,E2 3990.022} C_VEL
LIN {X 0,Y 682.338,Z 767.06,A -85,B 0,C 180,E1 3997.914,E2 3997.914} C_VEL
LIN {X 0,Y 682.544,Z 767.06,A -85,B 0,C 180,E1 4006.26,E2 4006.26} C_VEL
LIN {X 0,Y 682.86,Z 768.897,A -85,B 0,C 180,E1 4014.712,E2 4014.712} C_VEL
LIN {X 0,Y 699.364,Z 801.608,A -85,B 0,C 180,E1 4016.316,E2 4016.316} C_VEL
LIN {X 0,Y 697.735,Z 882.94,A -85,B 0,C 180,E1 4017.999,E2 4017.999} C_VEL
LIN {X 0,Y 694.29,Z 957.222,A -85,B 0,C 180,E1 4020.902,E2 4020.902} C_VEL
LIN {X 0,Y 690.319,Z 1027.292,A -85,B 0,C 180,E1 4025.116,E2 4025.116} C_VEL
LIN {X 0,Y 686.887,Z 1087.623,A -85,B 0,C 180,E1 4030.327,E2 4030.327} C_VEL
LIN {X 0,Y 684.461,Z 1135.909,A -85,B 0,C 180,E1 4036.223,E2 4036.223} C_VEL
LIN {X 0,Y 683.353,Z 1168.734,A -85,B 0,C 180,E1 4042.029,E2 4042.029} C_VEL
LIN {X 0,Y 683.162,Z 1188.503,A -85,B 0,C 180,E1 4047.457,E2 4047.457} C_VEL
LIN {X 0,Y 683.177,Z 1198.76,A -85,B 0,C 180,E1 4053.183,E2 4053.183} C_VEL
LIN {X 0,Y 682.998,Z 1197.888,A -85,B 0,C 180,E1 4059.588,E2 4059.588} C_VEL
LIN {X 0,Y 683.098,Z 1185.409,A -85,B 0,C 180,E1 4065.516,E2 4065.516} C_VEL
LIN {X 0,Y 683.657,Z 1161.011,A -85,B 0,C 180,E1 4071.471,E2 4071.471} C_VEL
LIN {X 0,Y 684.942,Z 1123.825,A -85,B 0,C 180,E1 4077.379,E2 4077.379} C_VEL
LIN {X 0,Y 687.717,Z 1072.069,A -85,B 0,C 180,E1 4083.106,E2 4083.106} C_VEL
LIN {X 0,Y 691.381,Z 1010.062,A -85,B 0,C 180,E1 4087.982,E2 4087.982} C_VEL
LIN {X 0,Y 695.334,Z 939.923,A -85,B 0,C 180,E1 4091.807,E2 4091.807} C_VEL
LIN {X 0,Y 698.516,Z 865.776,A -85,B 0,C 180,E1 4094.375,E2 4094.375} C_VEL
LIN {X 0,Y 698.084,Z 795.057,A -85,B 0,C 180,E1 4095.767,E2 4095.767} C_VEL
LIN {X 0,Y 682.388,Z 767.06,A -85,B 0,C 180,E1 4097.297,E2 4097.297} C_VEL
LIN {X 0,Y 682.268,Z 767.06,A -85,B 0,C 180,E1 4105.448,E2 4105.448} C_VEL
LIN {X 0,Y 682.342,Z 767.06,A -85,B 0,C 180,E1 4112.875,E2 4112.875} C_VEL
LIN {X 0,Y 682.488,Z 767.06,A -85,B 0,C 180,E1 4119.836,E2 4119.836} C_VEL
LIN {X 0,Y 683.421,Z 767.06,A -85,B 0,C 180,E1 4127.815,E2 4127.815} C_VEL
LIN {X 0,Y 683.137,Z 767.06,A -85,B 0,C 180,E1 4138.079,E2 4138.079} C_VEL
LIN {X 0,Y 682.984,Z 767.06,A -85,B 0,C 180,E1 4145.723,E2 4145.723} C_VEL
LIN {X 0,Y 682.83,Z 767.06,A -85,B 0,C 180,E1 4153.475,E2 4153.475} C_VEL
LIN {X 0,Y 682.585,Z 767.06,A -85,B 0,C 180,E1 4161.497,E2 4161.497} C_VEL
LIN {X 0,Y 681.97,Z 767.06,A -85,B 0,C 180,E1 4164.195,E2 4164.195} C_VEL
LIN {X 0,Y 674.471,Z 767.06,A -85,B 0,C 180,E1 4167.131,E2 4167.131} C_VEL
LIN {X 0,Y 674.347,Z 767.06,A -85,B 0,C 180,E1 4174.985,E2 4174.985} C_VEL
LIN {X 0,Y 674.217,Z 767.06,A -85,B 0,C 180,E1 4183.312,E2 4183.312} C_VEL
LIN {X 0,Y 674.218,Z 768.643,A -85,B 0,C 180,E1 4187.966,E2 4187.966} C_VEL
LIN {X 0,Y 693.694,Z 804.608,A -85,B 0,C 180,E1 4189.879,E2 4189.879} C_VEL
LIN {X 0,Y 691.387,Z 887.883,A -85,B 0,C 180,E1 4191.474,E2 4191.474} C_VEL
LIN {X 0,Y 687.636,Z 964.855,A -85,B 0,C 180,E1 4194.433,E2 4194.433} C_VEL
LIN {X 0,Y 683.474,Z 1033.973,A -85,B 0,C 180,E1 4198.571,E2 4198.571} C_VEL
LIN {X 0,Y 679.745,Z 1094.765,A -85,B 0,C 180,E1 4203.785,E2 4203.785} C_VEL
LIN {X 0,Y 677.442,Z 1143.521,A -85,B 0,C 180,E1 4209.696,E2 4209.696} C_VEL
LIN {X 0,Y 675.691,Z 1180.791,A -85,B 0,C 180,E1 4216.368,E2 4216.368} C_VEL
LIN {X 0,Y 675.073,Z 1202.161,A -85,B 0,C 180,E1 4222.901,E2 4222.901} C_VEL
LIN {X 0,Y 675.234,Z 1209.402,A -85,B 0,C 180,E1 4228.068,E2 4228.068} C_VEL
LIN {X 0,Y 675.209,Z 1206.829,A -85,B 0,C 180,E1 4234.507,E2 4234.507} C_VEL
LIN {X 0,Y 675.217,Z 1192.193,A -85,B 0,C 180,E1 4240.676,E2 4240.676} C_VEL
LIN {X 0,Y 675.914,Z 1164.616,A -85,B 0,C 180,E1 4246.914,E2 4246.914} C_VEL
LIN {X 0,Y 677.618,Z 1125.845,A -85,B 0,C 180,E1 4252.706,E2 4252.706} C_VEL
LIN {X 0,Y 680.725,Z 1072.386,A -85,B 0,C 180,E1 4258.363,E2 4258.363} C_VEL
LIN {X 0,Y 685.129,Z 1007.497,A -85,B 0,C 180,E1 4263.21,E2 4263.21} C_VEL
LIN {X 0,Y 689.434,Z 936.309,A -85,B 0,C 180,E1 4266.834,E2 4266.834} C_VEL
LIN {X 0,Y 692.688,Z 861.387,A -85,B 0,C 180,E1 4269.178,E2 4269.178} C_VEL
LIN {X 0,Y 692.07,Z 799.366,A -85,B 0,C 180,E1 4270.304,E2 4270.304} C_VEL
LIN {X 0,Y 674.858,Z 767.06,A -85,B 0,C 180,E1 4272.199,E2 4272.199} C_VEL
LIN {X 0,Y 674.663,Z 767.06,A -85,B 0,C 180,E1 4281.825,E2 4281.825} C_VEL
LIN {X 0,Y 674.469,Z 767.06,A -85,B 0,C 180,E1 4289.95,E2 4289.95} C_VEL
LIN {X 0,Y 674.069,Z 767.06,A -85,B 0,C 180,E1 4296.823,E2 4296.823} C_VEL
LIN {X 0,Y 674.504,Z 767.06,A -85,B 0,C 180,E1 4303.687,E2 4303.687} C_VEL
LIN {X 0,Y 674.53,Z 767.06,A -85,B 0,C 180,E1 4311.608,E2 4311.608} C_VEL
LIN {X 0,Y 675.092,Z 767.06,A -85,B 0,C 180,E1 4318.081,E2 4318.081} C_VEL
LIN {X 0,Y 675.032,Z 767.06,A -85,B 0,C 180,E1 4325.817,E2 4325.817} C_VEL
LIN {X 0,Y 674.764,Z 767.06,A -85,B 0,C 180,E1 4333.666,E2 4333.666} C_VEL
LIN {X 0,Y 674.442,Z 767.06,A -85,B 0,C 180,E1 4341.797,E2 4341.797} C_VEL
LIN {X 0,Y 674.319,Z 767.06,A -85,B 0,C 180,E1 4350.421,E2 4350.421} C_VEL
LIN {X 0,Y 674.258,Z 767.06,A -85,B 0,C 180,E1 4358.235,E2 4358.235} C_VEL
LIN {X 0,Y 674.389,Z 767.06,A -85,B 0,C 180,E1 4366.989,E2 4366.989} C_VEL
LIN {X 0,Y 674.88,Z 768.66,A -85,B 0,C 180,E1 4374.112,E2 4374.112} C_VEL
LIN {X 0,Y 693.301,Z 805.96,A -85,B 0,C 180,E1 4375.957,E2 4375.957} C_VEL
LIN {X 0,Y 691.26,Z 885.979,A -85,B 0,C 180,E1 4377.676,E2 4377.676} C_VEL
LIN {X 0,Y 687.402,Z 960.653,A -85,B 0,C 180,E1 4380.674,E2 4380.674} C_VEL
LIN {X 0,Y 682.965,Z 1030.105,A -85,B 0,C 180,E1 4384.961,E2 4384.961} C_VEL
LIN {X 0,Y 679.155,Z 1089.902,A -85,B 0,C 180,E1 4390.264,E2 4390.264} C_VEL
LIN {X 0,Y 676.553,Z 1137.473,A -85,B 0,C 180,E1 4396.224,E2 4396.224} C_VEL
LIN {X 0,Y 675.322,Z 1170.56,A -85,B 0,C 180,E1 4402.259,E2 4402.259} C_VEL
LIN {X 0,Y 674.888,Z 1190.323,A -85,B 0,C 180,E1 4408.07,E2 4408.07} C_VEL
LIN {X 0,Y 675.154,Z 1198.816,A -85,B 0,C 180,E1 4413.221,E2 4413.221} C_VEL
LIN {X 0,Y 674.961,Z 1197.802,A -85,B 0,C 180,E1 4419.703,E2 4419.703} C_VEL
LIN {X 0,Y 675.085,Z 1185.377,A -85,B 0,C 180,E1 4425.64,E2 4425.64} C_VEL
LIN {X 0,Y 675.739,Z 1161.974,A -85,B 0,C 180,E1 4431.472,E2 4431.472} C_VEL
LIN {X 0,Y 677.137,Z 1124.506,A -85,B 0,C 180,E1 4437.542,E2 4437.542} C_VEL
LIN {X 0,Y 680.204,Z 1072.909,A -85,B 0,C 180,E1 4443.352,E2 4443.352} C_VEL
LIN {X 0,Y 684.292,Z 1010.078,A -85,B 0,C 180,E1 4448.353,E2 4448.353} C_VEL
LIN {X 0,Y 688.683,Z 940.248,A -85,B 0,C 180,E1 4452.193,E2 4452.193} C_VEL
LIN {X 0,Y 692.201,Z 866.398,A -85,B 0,C 180,E1 4454.774,E2 4454.774} C_VEL
LIN {X 0,Y 691.977,Z 798.428,A -85,B 0,C 180,E1 4456.145,E2 4456.145} C_VEL
LIN {X 0,Y 674.256,Z 767.06,A -85,B 0,C 180,E1 4457.965,E2 4457.965} C_VEL
LIN {X 0,Y 674.303,Z 767.06,A -85,B 0,C 180,E1 4465.174,E2 4465.174} C_VEL
LIN {X 0,Y 674.365,Z 767.06,A -85,B 0,C 180,E1 4472.657,E2 4472.657} C_VEL
LIN {X 0,Y 674.509,Z 767.06,A -85,B 0,C 180,E1 4479.586,E2 4479.586} C_VEL
LIN {X 0,Y 675.391,Z 767.06,A -85,B 0,C 180,E1 4487.667,E2 4487.667} C_VEL
LIN {X 0,Y 675.147,Z 767.06,A -85,B 0,C 180,E1 4498.056,E2 4498.056} C_VEL
LIN {X 0,Y 674.949,Z 767.06,A -85,B 0,C 180,E1 4505.791,E2 4505.791} C_VEL
LIN {X 0,Y 674.744,Z 767.06,A -85,B 0,C 180,E1 4513.64,E2 4513.64} C_VEL
LIN {X 0,Y 674.486,Z 767.06,A -85,B 0,C 180,E1 4521.768,E2 4521.768} C_VEL
LIN {X 0,Y 674.471,Z 767.06,A -85,B 0,C 180,E1 4527.131,E2 4527.131} C_VEL
LIN {X 0,Y 666.352,Z 767.06,A -85,B 0,C 180,E1 4530.1,E2 4530.1} C_VEL
LIN {X 0,Y 666.063,Z 767.06,A -85,B 0,C 180,E1 4538.759,E2 4538.759} C_VEL
LIN {X 0,Y 666.288,Z 768.246,A -85,B 0,C 180,E1 4547.343,E2 4547.343} C_VEL
LIN {X 0,Y 687.567,Z 808.401,A -85,B 0,C 180,E1 4549.499,E2 4549.499} C_VEL
LIN {X 0,Y 684.941,Z 890.689,A -85,B 0,C 180,E1 4551.131,E2 4551.131} C_VEL
LIN {X 0,Y 680.771,Z 967.306,A -85,B 0,C 180,E1 4554.147,E2 4554.147} C_VEL
LIN {X 0,Y 676.142,Z 1036.924,A -85,B 0,C 180,E1 4558.413,E2 4558.413} C_VEL
LIN {X 0,Y 672.11,Z 1096.672,A -85,B 0,C 180,E1 4563.661,E2 4563.661} C_VEL
LIN {X 0,Y 669.379,Z 1146.192,A -85,B 0,C 180,E1 4569.848,E2 4569.848} C_VEL
LIN {X 0,Y 667.627,Z 1182.147,A -85,B 0,C 180,E1 4576.535,E2 4576.535} C_VEL
LIN {X 0,Y 667.106,Z 1202.161,A -85,B 0,C 180,E1 4582.816,E2 4582.816} C_VEL
LIN {X 0,Y 667.238,Z 1209.402,A -85,B 0,C 180,E1 4588.044,E2 4588.044} C_VEL
LIN {X 0,Y 667.181,Z 1206.826,A -85,B 0,C 180,E1 4594.561,E2 4594.561} C_VEL
LIN {X 0,Y 667.201,Z 1192.193,A -85,B 0,C 180,E1 4600.806,E2 4600.806} C_VEL
LIN {X 0,Y 667.995,Z 1164.885,A -85,B 0,C 180,E1 4607.069,E2 4607.069} C_VEL
LIN {X 0,Y 669.806,Z 1125.844,A -85,B 0,C 180,E1 4612.986,E2 4612.986} C_VEL
LIN {X 0,Y 673.367,Z 1072.386,A -85,B 0,C 180,E1 4618.702,E2 4618.702} C_VEL
LIN {X 0,Y 678.154,Z 1007.5,A -85,B 0,C 180,E1 4623.597,E2 4623.597} C_VEL
LIN {X 0,Y 682.905,Z 936.264,A -85,B 0,C 180,E1 4627.248,E2 4627.248} C_VEL
LIN {X 0,Y 686.387,Z 863.091,A -85,B 0,C 180,E1 4629.563,E2 4629.563} C_VEL
LIN {X 0,Y 686.048,Z 802.806,A -85,B 0,C 180,E1 4630.685,E2 4630.685} C_VEL
LIN {X 0,Y 666.753,Z 767.06,A -85,B 0,C 180,E1 4632.822,E2 4632.822} C_VEL
LIN {X 0,Y 666.687,Z 767.06,A -85,B 0,C 180,E1 4641.694,E2 4641.694} C_VEL
LIN {X 0,Y 666.472,Z 767.06,A -85,B 0,C 180,E1 4649.212,E2 4649.212} C_VEL
LIN {X 0,Y 666.116,Z 767.06,A -85,B 0,C 180,E1 4656.53,E2 4656.53} C_VEL
LIN {X 0,Y 666.569,Z 767.06,A -85,B 0,C 180,E1 4663.487,E2 4663.487} C_VEL
LIN {X 0,Y 666.495,Z 767.06,A -85,B 0,C 180,E1 4671.773,E2 4671.773} C_VEL
LIN {X 0,Y 667.095,Z 767.06,A -85,B 0,C 180,E1 4678.058,E2 4678.058} C_VEL
LIN {X 0,Y 666.983,Z 767.06,A -85,B 0,C 180,E1 4685.887,E2 4685.887} C_VEL
LIN {X 0,Y 666.68,Z 767.06,A -85,B 0,C 180,E1 4693.835,E2 4693.835} C_VEL
LIN {X 0,Y 666.327,Z 767.06,A -85,B 0,C 180,E1 4702.076,E2 4702.076} C_VEL
LIN {X 0,Y 666.533,Z 767.06,A -85,B 0,C 180,E1 4709.309,E2 4709.309} C_VEL
LIN {X 0,Y 666.261,Z 767.06,A -85,B 0,C 180,E1 4718.26,E2 4718.26} C_VEL
LIN {X 0,Y 666.45,Z 767.06,A -85,B 0,C 180,E1 4726.055,E2 4726.055} C_VEL
LIN {X 0,Y 666.849,Z 768.676,A -85,B 0,C 180,E1 4733.492,E2 4733.492} C_VEL
LIN {X 0,Y 687.185,Z 808.664,A -85,B 0,C 180,E1 4735.567,E2 4735.567} C_VEL
LIN {X 0,Y 684.784,Z 888.361,A -85,B 0,C 180,E1 4737.333,E2 4737.333} C_VEL
LIN {X 0,Y 680.577,Z 962.189,A -85,B 0,C 180,E1 4740.351,E2 4740.351} C_VEL
LIN {X 0,Y 675.738,Z 1031.108,A -85,B 0,C 180,E1 4744.675,E2 4744.675} C_VEL
LIN {X 0,Y 671.539,Z 1091.124,A -85,B 0,C 180,E1 4750.087,E2 4750.087} C_VEL
LIN {X 0,Y 668.726,Z 1137.962,A -85,B 0,C 180,E1 4756.06,E2 4756.06} C_VEL
LIN {X 0,Y 667.379,Z 1170.86,A -85,B 0,C 180,E1 4762.166,E2 4762.166} C_VEL
LIN {X 0,Y 666.896,Z 1190.492,A -85,B 0,C 180,E1 4768.047,E2 4768.047} C_VEL
LIN {X 0,Y 667.132,Z 1198.87,A -85,B 0,C 180,E1 4773.26,E2 4773.26} C_VEL
LIN {X 0,Y 666.928,Z 1197.715,A -85,B 0,C 180,E1 4779.821,E2 4779.821} C_VEL
LIN {X 0,Y 667.077,Z 1185.152,A -85,B 0,C 180,E1 4785.833,E2 4785.833} C_VEL
LIN {X 0,Y 667.723,Z 1161.357,A -85,B 0,C 180,E1 4791.783,E2 4791.783} C_VEL
LIN {X 0,Y 669.419,Z 1123.925,A -85,B 0,C 180,E1 4797.887,E2 4797.887} C_VEL
LIN {X 0,Y 672.708,Z 1073.424,A -85,B 0,C 180,E1 4803.633,E2 4803.633} C_VEL
LIN {X 0,Y 677.223,Z 1009.772,A -85,B 0,C 180,E1 4808.754,E2 4808.754} C_VEL
LIN {X 0,Y 682.082,Z 939.964,A -85,B 0,C 180,E1 4812.614,E2 4812.614} C_VEL
LIN {X 0,Y 685.926,Z 866.42,A -85,B 0,C 180,E1 4815.196,E2 4815.196} C_VEL
LIN {X 0,Y 686.03,Z 802.134,A -85,B 0,C 180,E1 4816.516,E2 4816.516} C_VEL
LIN {X 0,Y 666.181,Z 767.06,A -85,B 0,C 180,E1 4818.639,E2 4818.639} C_VEL
LIN {X 0,Y 666.223,Z 767.06,A -85,B 0,C 180,E1 4826.186,E2 4826.186} C_VEL
LIN {X 0,Y 666.257,Z 767.06,A -85,B 0,C 180,E1 4834.038,E2 4834.038} C_VEL
LIN {X 0,Y 666.323,Z 767.06,A -85,B 0,C 180,E1 4840.824,E2 4840.824} C_VEL
LIN {X 0,Y 667.405,Z 767.06,A -85,B 0,C 180,E1 4848.848,E2 4848.848} C_VEL
LIN {X 0,Y 667.15,Z 767.06,A -85,B 0,C 180,E1 4858.033,E2 4858.033} C_VEL
LIN {X 0,Y 666.9,Z 767.06,A -85,B 0,C 180,E1 4865.862,E2 4865.862} C_VEL
LIN {X 0,Y 666.665,Z 767.06,A -85,B 0,C 180,E1 4873.809,E2 4873.809} C_VEL
LIN {X 0,Y 666.37,Z 767.06,A -85,B 0,C 180,E1 4882.047,E2 4882.047} C_VEL
LIN {X 0,Y 666.352,Z 767.06,A -85,B 0,C 180,E1 4890.1,E2 4890.1} C_VEL
LIN {X 0,Y 658.022,Z 767.06,A -85,B 0,C 180,E1 4893.074,E2 4893.074} C_VEL
LIN {X 0,Y 657.9,Z 767.06,A -85,B 0,C 180,E1 4899.448,E2 4899.448} C_VEL
LIN {X 0,Y 658.397,Z 767.717,A -85,B 0,C 180,E1 4906.699,E2 4906.699} C_VEL
LIN {X 0,Y 681.515,Z 813.426,A -85,B 0,C 180,E1 4909.131,E2 4909.131} C_VEL
LIN {X 0,Y 678.392,Z 894.34,A -85,B 0,C 180,E1 4910.803,E2 4910.803} C_VEL
LIN {X 0,Y 673.9,Z 970.36,A -85,B 0,C 180,E1 4913.886,E2 4913.886} C_VEL
LIN {X 0,Y 668.791,Z 1039.724,A -85,B 0,C 180,E1 4918.244,E2 4918.244} C_VEL
LIN {X 0,Y 664.428,Z 1098.785,A -85,B 0,C 180,E1 4923.571,E2 4923.571} C_VEL
LIN {X 0,Y 661.574,Z 1146.966,A -85,B 0,C 180,E1 4929.723,E2 4929.723} C_VEL
LIN {X 0,Y 659.727,Z 1182.148,A -85,B 0,C 180,E1 4936.371,E2 4936.371} C_VEL
LIN {X 0,Y 659.142,Z 1202.161,A -85,B 0,C 180,E1 4942.729,E2 4942.729} C_VEL
LIN {X 0,Y 659.258,Z 1209.402,A -85,B 0,C 180,E1 4948.021,E2 4948.021} C_VEL
LIN {X 0,Y 659.182,Z 1206.824,A -85,B 0,C 180,E1 4954.616,E2 4954.616} C_VEL
LIN {X 0,Y 659.188,Z 1192.193,A -85,B 0,C 180,E1 4960.939,E2 4960.939} C_VEL
LIN {X 0,Y 660.084,Z 1165.68,A -85,B 0,C 180,E1 4967.125,E2 4967.125} C_VEL
LIN {X 0,Y 662.042,Z 1127.193,A -85,B 0,C 180,E1 4973.093,E2 4973.093} C_VEL
LIN {X 0,Y 665.917,Z 1073.59,A -85,B 0,C 180,E1 4978.937,E2 4978.937} C_VEL
LIN {X 0,Y 671.055,Z 1009.585,A -85,B 0,C 180,E1 4983.854,E2 4983.854} C_VEL
LIN {X 0,Y 676.129,Z 940.026,A -85,B 0,C 180,E1 4987.507,E2 4987.507} C_VEL
LIN {X 0,Y 679.964,Z 866.791,A -85,B 0,C 180,E1 4989.914,E2 4989.914} C_VEL
LIN {X 0,Y 680.157,Z 806.33,A -85,B 0,C 180,E1 4991.065,E2 4991.065} C_VEL
LIN {X 0,Y 658.556,Z 767.06,A -85,B 0,C 180,E1 4993.505,E2 4993.505} C_VEL
LIN {X 0,Y 658.628,Z 767.06,A -85,B 0,C 180,E1 5002.59,E2 5002.59} C_VEL
LIN {X 0,Y 658.429,Z 767.06,A -85,B 0,C 180,E1 5010.325,E2 5010.325} C_VEL
LIN {X 0,Y 658.014,Z 767.06,A -85,B 0,C 180,E1 5017.658,E2 5017.658} C_VEL
LIN {X 0,Y 658.28,Z 767.06,A -85,B 0,C 180,E1 5024.647,E2 5024.647} C_VEL
LIN {X 0,Y 658.589,Z 767.06,A -85,B 0,C 180,E1 5031.403,E2 5031.403} C_VEL
LIN {X 0,Y 659.106,Z 767.06,A -85,B 0,C 180,E1 5038.035,E2 5038.035} C_VEL
LIN {X 0,Y 658.935,Z 767.06,A -85,B 0,C 180,E1 5045.959,E2 5045.959} C_VEL
LIN {X 0,Y 658.626,Z 767.06,A -85,B 0,C 180,E1 5054.008,E2 5054.008} C_VEL
LIN {X 0,Y 658.233,Z 767.06,A -85,B 0,C 180,E1 5062.362,E2 5062.362} C_VEL
LIN {X 0,Y 658.273,Z 767.06,A -85,B 0,C 180,E1 5070.248,E2 5070.248} C_VEL
LIN {X 0,Y 658.341,Z 767.06,A -85,B 0,C 180,E1 5077.648,E2 5077.648} C_VEL
LIN {X 0,Y 658.349,Z 767.06,A -85,B 0,C 180,E1 5086.552,E2 5086.552} C_VEL
LIN {X 0,Y 658.795,Z 768.461,A -85,B 0,C 180,E1 5092.844,E2 5092.844} C_VEL
LIN {X 0,Y 681.097,Z 811.396,A -85,B 0,C 180,E1 5095.173,E2 5095.173} C_VEL
LIN {X 0,Y 678.381,Z 889.545,A -85,B 0,C 180,E1 5096.943,E2 5096.943} C_VEL
LIN {X 0,Y 673.736,Z 963.809,A -85,B 0,C 180,E1 5100.028,E2 5100.028} C_VEL
LIN {X 0,Y 668.513,Z 1032.113,A -85,B 0,C 180,E1 5104.381,E2 5104.381} C_VEL
LIN {X 0,Y 664.073,Z 1091.071,A -85,B 0,C 180,E1 5109.768,E2 5109.768} C_VEL
LIN {X 0,Y 660.922,Z 1138.45,A -85,B 0,C 180,E1 5115.892,E2 5115.892} C_VEL
LIN {X 0,Y 659.443,Z 1171.159,A -85,B 0,C 180,E1 5122.071,E2 5122.071} C_VEL
LIN {X 0,Y 658.912,Z 1190.66,A -85,B 0,C 180,E1 5128.024,E2 5128.024} C_VEL
LIN {X 0,Y 659.132,Z 1198.923,A -85,B 0,C 180,E1 5133.299,E2 5133.299} C_VEL
LIN {X 0,Y 658.9,Z 1197.629,A -85,B 0,C 180,E1 5139.942,E2 5139.942} C_VEL
LIN {X 0,Y 659.051,Z 1184.92,A -85,B 0,C 180,E1 5146.031,E2 5146.031} C_VEL
LIN {X 0,Y 659.818,Z 1161.049,A -85,B 0,C 180,E1 5152.038,E2 5152.038} C_VEL
LIN {X 0,Y 661.623,Z 1124.836,A -85,B 0,C 180,E1 5158.028,E2 5158.028} C_VEL
LIN {X 0,Y 665.225,Z 1073.592,A -85,B 0,C 180,E1 5163.955,E2 5163.955} C_VEL
LIN {X 0,Y 670.22,Z 1009.701,A -85,B 0,C 180,E1 5169.146,E2 5169.146} C_VEL
LIN {X 0,Y 675.458,Z 940.933,A -85,B 0,C 180,E1 5172.987,E2 5172.987} C_VEL
LIN {X 0,Y 679.633,Z 867.679,A -85,B 0,C 180,E1 5175.593,E2 5175.593} C_VEL
LIN {X 0,Y 679.862,Z 805.183,A -85,B 0,C 180,E1 5176.92,E2 5176.92} C_VEL
LIN {X 0,Y 658.191,Z 767.06,A -85,B 0,C 180,E1 5179.236,E2 5179.236} C_VEL
LIN {X 0,Y 658.246,Z 767.06,A -85,B 0,C 180,E1 5187.237,E2 5187.237} C_VEL
LIN {X 0,Y 658.402,Z 767.06,A -85,B 0,C 180,E1 5195.479,E2 5195.479} C_VEL
LIN {X 0,Y 658.958,Z 767.06,A -85,B 0,C 180,E1 5204.636,E2 5204.636} C_VEL
LIN {X 0,Y 658.656,Z 767.06,A -85,B 0,C 180,E1 5211.378,E2 5211.378} C_VEL
LIN {X 0,Y 659.16,Z 767.06,A -85,B 0,C 180,E1 5218.009,E2 5218.009} C_VEL
LIN {X 0,Y 658.854,Z 767.06,A -85,B 0,C 180,E1 5225.933,E2 5225.933} C_VEL
LIN {X 0,Y 658.614,Z 767.06,A -85,B 0,C 180,E1 5233.981,E2 5233.981} C_VEL
LIN {X 0,Y 658.305,Z 767.06,A -85,B 0,C 180,E1 5242.331,E2 5242.331} C_VEL
LIN {X 0,Y 658.327,Z 767.06,A -85,B 0,C 180,E1 5250.249,E2 5250.249} C_VEL
LIN {X 0,Y 658.022,Z 767.06,A -85,B 0,C 180,E1 5253.074,E2 5253.074} C_VEL
LIN {X 0,Y 650.247,Z 767.06,A -85,B 0,C 180,E1 5256.114,E2 5256.114} C_VEL
LIN {X 0,Y 650.364,Z 767.834,A -85,B 0,C 180,E1 5266.03,E2 5266.03} C_VEL
LIN {X 0,Y 675.444,Z 816.173,A -85,B 0,C 180,E1 5268.723,E2 5268.723} C_VEL
LIN {X 0,Y 672.043,Z 896.143,A -85,B 0,C 180,E1 5270.423,E2 5270.423} C_VEL
LIN {X 0,Y 667.143,Z 971.726,A -85,B 0,C 180,E1 5273.54,E2 5273.54} C_VEL
LIN {X 0,Y 661.6,Z 1040.754,A -85,B 0,C 180,E1 5277.944,E2 5277.944} C_VEL
LIN {X 0,Y 656.855,Z 1099.822,A -85,B 0,C 180,E1 5283.36,E2 5283.36} C_VEL
LIN {X 0,Y 653.782,Z 1147.488,A -85,B 0,C 180,E1 5289.554,E2 5289.554} C_VEL
LIN {X 0,Y 651.85,Z 1182.149,A -85,B 0,C 180,E1 5296.203,E2 5296.203} C_VEL
LIN {X 0,Y 651.178,Z 1202.16,A -85,B 0,C 180,E1 5302.639,E2 5302.639} C_VEL
LIN {X 0,Y 651.261,Z 1209.402,A -85,B 0,C 180,E1 5307.996,E2 5307.996} C_VEL
LIN {X 0,Y 651.154,Z 1206.821,A -85,B 0,C 180,E1 5314.673,E2 5314.673} C_VEL
LIN {X 0,Y 651.179,Z 1192.192,A -85,B 0,C 180,E1 5321.075,E2 5321.075} C_VEL
LIN {X 0,Y 652.18,Z 1165.682,A -85,B 0,C 180,E1 5327.339,E2 5327.339} C_VEL
LIN {X 0,Y 654.308,Z 1127.814,A -85,B 0,C 180,E1 5333.299,E2 5333.299} C_VEL
LIN {X 0,Y 658.468,Z 1074.75,A -85,B 0,C 180,E1 5339.182,E2 5339.182} C_VEL
LIN {X 0,Y 664.119,Z 1010.301,A -85,B 0,C 180,E1 5344.205,E2 5344.205} C_VEL
LIN {X 0,Y 669.62,Z 940.453,A -85,B 0,C 180,E1 5347.915,E2 5347.915} C_VEL
LIN {X 0,Y 673.757,Z 867.525,A -85,B 0,C 180,E1 5350.336,E2 5350.336} C_VEL
LIN {X 0,Y 673.894,Z 809.062,A -85,B 0,C 180,E1 5351.493,E2 5351.493} C_VEL
LIN {X 0,Y 650.355,Z 767.06,A -85,B 0,C 180,E1 5354.12,E2 5354.12} C_VEL
LIN {X 0,Y 650.55,Z 767.06,A -85,B 0,C 180,E1 5361.855,E2 5361.855} C_VEL
LIN {X 0,Y 650.439,Z 767.06,A -85,B 0,C 180,E1 5369.923,E2 5369.923} C_VEL
LIN {X 0,Y 650.009,Z 767.06,A -85,B 0,C 180,E1 5377.368,E2 5377.368} C_VEL
LIN {X 0,Y 650.332,Z 767.06,A -85,B 0,C 180,E1 5384.455,E2 5384.455} C_VEL
LIN {X 0,Y 650.353,Z 767.06,A -85,B 0,C 180,E1 5392.289,E2 5392.289} C_VEL
LIN {X 0,Y 651.108,Z 767.06,A -85,B 0,C 180,E1 5398.011,E2 5398.011} C_VEL
LIN {X 0,Y 650.891,Z 767.06,A -85,B 0,C 180,E1 5406.033,E2 5406.033} C_VEL
LIN {X 0,Y 650.408,Z 767.06,A -85,B 0,C 180,E1 5414.634,E2 5414.634} C_VEL
LIN {X 0,Y 650.11,Z 767.06,A -85,B 0,C 180,E1 5422.876,E2 5422.876} C_VEL
LIN {X 0,Y 650.317,Z 767.06,A -85,B 0,C 180,E1 5430.114,E2 5430.114} C_VEL
LIN {X 0,Y 650.096,Z 767.06,A -85,B 0,C 180,E1 5438.61,E2 5438.61} C_VEL
LIN {X 0,Y 650.23,Z 767.06,A -85,B 0,C 180,E1 5447.313,E2 5447.313} C_VEL
LIN {X 0,Y 650.773,Z 768.984,A -85,B 0,C 180,E1 5452.187,E2 5452.187} C_VEL
LIN {X 0,Y 675.025,Z 814.365,A -85,B 0,C 180,E1 5454.777,E2 5454.777} C_VEL
LIN {X 0,Y 671.901,Z 892.762,A -85,B 0,C 180,E1 5456.615,E2 5456.615} C_VEL
LIN {X 0,Y 666.88,Z 965.991,A -85,B 0,C 180,E1 5459.73,E2 5459.73} C_VEL
LIN {X 0,Y 661.191,Z 1034.219,A -85,B 0,C 180,E1 5464.168,E2 5464.168} C_VEL
LIN {X 0,Y 656.336,Z 1093.386,A -85,B 0,C 180,E1 5469.699,E2 5469.699} C_VEL
LIN {X 0,Y 653.004,Z 1140.015,A -85,B 0,C 180,E1 5475.889,E2 5475.889} C_VEL
LIN {X 0,Y 651.517,Z 1171.365,A -85,B 0,C 180,E1 5481.951,E2 5481.951} C_VEL
LIN {X 0,Y 650.919,Z 1190.828,A -85,B 0,C 180,E1 5487.999,E2 5487.999} C_VEL
LIN {X 0,Y 651.11,Z 1198.977,A -85,B 0,C 180,E1 5493.34,E2 5493.34} C_VEL
LIN {X 0,Y 650.877,Z 1197.543,A -85,B 0,C 180,E1 5500.065,E2 5500.065} C_VEL
LIN {X 0,Y 651.052,Z 1184.689,A -85,B 0,C 180,E1 5506.233,E2 5506.233} C_VEL
LIN {X 0,Y 651.869,Z 1161.694,A -85,B 0,C 180,E1 5512.11,E2 5512.11} C_VEL
LIN {X 0,Y 653.872,Z 1125.042,A -85,B 0,C 180,E1 5518.274,E2 5518.274} C_VEL
LIN {X 0,Y 657.732,Z 1074.42,A -85,B 0,C 180,E1 5524.215,E2 5524.215} C_VEL
LIN {X 0,Y 663.09,Z 1011.9,A -85,B 0,C 180,E1 5529.394,E2 5529.394} C_VEL
LIN {X 0,Y 668.854,Z 942.06,A -85,B 0,C 180,E1 5533.361,E2 5533.361} C_VEL
LIN {X 0,Y 673.345,Z 869.268,A -85,B 0,C 180,E1 5535.989,E2 5535.989} C_VEL
LIN {X 0,Y 673.805,Z 808.579,A -85,B 0,C 180,E1 5537.319,E2 5537.319} C_VEL
LIN {X 0,Y 650.232,Z 767.06,A -85,B 0,C 180,E1 5539.927,E2 5539.927} C_VEL
LIN {X 0,Y 650.368,Z 767.06,A -85,B 0,C 180,E1 5548.332,E2 5548.332} C_VEL
LIN {X 0,Y 650.63,Z 767.06,A -85,B 0,C 180,E1 5557.362,E2 5557.362} C_VEL
LIN {X 0,Y 651.329,Z 767.06,A -85,B 0,C 180,E1 5567.204,E2 5567.204} C_VEL
LIN {X 0,Y 651.336,Z 767.06,A -85,B 0,C 180,E1 5576.776,E2 5576.776} C_VEL
LIN {X 0,Y 650.81,Z 767.06,A -85,B 0,C 180,E1 5586.007,E2 5586.007} C_VEL
LIN {X 0,Y 650.391,Z 767.06,A -85,B 0,C 180,E1 5594.613,E2 5594.613} C_VEL
LIN {X 0,Y 650.208,Z 767.06,A -85,B 0,C 180,E1 5602.625,E2 5602.625} C_VEL
LIN {X 0,Y 650.369,Z 767.06,A -85,B 0,C 180,E1 5610.08,E2 5610.08} C_VEL
LIN {X 0,Y 650.247,Z 767.06,A -85,B 0,C 180,E1 5616.114,E2 5616.114} C_VEL
LIN {X 0,Y 641.881,Z 767.06,A -85,B 0,C 180,E1 5619.178,E2 5619.178} C_VEL
LIN {X 0,Y 642.456,Z 768.451,A -85,B 0,C 180,E1 5625.356,E2 5625.356} C_VEL
LIN {X 0,Y 669.408,Z 819.333,A -85,B 0,C 180,E1 5628.317,E2 5628.317} C_VEL
LIN {X 0,Y 665.602,Z 899.443,A -85,B 0,C 180,E1 5630.088,E2 5630.088} C_VEL
LIN {X 0,Y 660.321,Z 973.772,A -85,B 0,C 180,E1 5633.224,E2 5633.224} C_VEL
LIN {X 0,Y 654.456,Z 1041.813,A -85,B 0,C 180,E1 5637.642,E2 5637.642} C_VEL
LIN {X 0,Y 649.348,Z 1100.381,A -85,B 0,C 180,E1 5643.092,E2 5643.092} C_VEL
LIN {X 0,Y 645.832,Z 1149.343,A -85,B 0,C 180,E1 5649.592,E2 5649.592} C_VEL
LIN {X 0,Y 643.771,Z 1183.506,A -85,B 0,C 180,E1 5656.373,E2 5656.373} C_VEL
LIN {X 0,Y 643.246,Z 1202.16,A -85,B 0,C 180,E1 5662.548,E2 5662.548} C_VEL
LIN {X 0,Y 643.271,Z 1209.402,A -85,B 0,C 180,E1 5667.972,E2 5667.972} C_VEL
LIN {X 0,Y 643.128,Z 1206.818,A -85,B 0,C 180,E1 5674.732,E2 5674.732} C_VEL
LIN {X 0,Y 643.18,Z 1192.192,A -85,B 0,C 180,E1 5681.214,E2 5681.214} C_VEL
LIN {X 0,Y 644.254,Z 1166.75,A -85,B 0,C 180,E1 5687.346,E2 5687.346} C_VEL
LIN {X 0,Y 646.539,Z 1129.462,A -85,B 0,C 180,E1 5693.369,E2 5693.369} C_VEL
LIN {X 0,Y 650.974,Z 1076.782,A -85,B 0,C 180,E1 5699.348,E2 5699.348} C_VEL
LIN {X 0,Y 656.982,Z 1012.99,A -85,B 0,C 180,E1 5704.436,E2 5704.436} C_VEL
LIN {X 0,Y 662.987,Z 942.946,A -85,B 0,C 180,E1 5708.242,E2 5708.242} C_VEL
LIN {X 0,Y 667.651,Z 867.505,A -85,B 0,C 180,E1 5710.783,E2 5710.783} C_VEL
LIN {X 0,Y 668.126,Z 812.821,A -85,B 0,C 180,E1 5711.878,E2 5711.878} C_VEL
LIN {X 0,Y 642.176,Z 767.06,A -85,B 0,C 180,E1 5714.802,E2 5714.802} C_VEL
LIN {X 0,Y 642.555,Z 767.06,A -85,B 0,C 180,E1 5723.006,E2 5723.006} C_VEL
LIN {X 0,Y 642.436,Z 767.06,A -85,B 0,C 180,E1 5731.067,E2 5731.067} C_VEL
LIN {X 0,Y 642.424,Z 767.06,A -85,B 0,C 180,E1 5739.993,E2 5739.993} C_VEL
LIN {X 0,Y 642.728,Z 767.06,A -85,B 0,C 180,E1 5748.442,E2 5748.442} C_VEL
LIN {X 0,Y 643.132,Z 767.06,A -85,B 0,C 180,E1 5757.986,E2 5757.986} C_VEL
LIN {X 0,Y 642.867,Z 767.06,A -85,B 0,C 180,E1 5766.109,E2 5766.109} C_VEL
LIN {X 0,Y 642.511,Z 767.06,A -85,B 0,C 180,E1 5774.366,E2 5774.366} C_VEL
LIN {X 0,Y 642.109,Z 767.06,A -85,B 0,C 180,E1 5782.956,E2 5782.956} C_VEL
LIN {X 0,Y 642.219,Z 767.06,A -85,B 0,C 180,E1 5790.534,E2 5790.534} C_VEL
LIN {X 0,Y 642.056,Z 767.06,A -85,B 0,C 180,E1 5798.778,E2 5798.778} C_VEL
LIN {X 0,Y 642.378,Z 767.06,A -85,B 0,C 180,E1 5806.091,E2 5806.091} C_VEL
LIN {X 0,Y 642.532,Z 768.515,A -85,B 0,C 180,E1 5811.472,E2 5811.472} C_VEL
LIN {X 0,Y 668.986,Z 816.657,A -85,B 0,C 180,E1 5814.363,E2 5814.363} C_VEL
LIN {X 0,Y 665.549,Z 894.022,A -85,B 0,C 180,E1 5816.213,E2 5816.213} C_VEL
LIN {X 0,Y 660.068,Z 967.956,A -85,B 0,C 180,E1 5819.415,E2 5819.415} C_VEL
LIN {X 0,Y 653.905,Z 1036.321,A -85,B 0,C 180,E1 5823.951,E2 5823.951} C_VEL
LIN {X 0,Y 648.623,Z 1095.453,A -85,B 0,C 180,E1 5829.605,E2 5829.605} C_VEL
LIN {X 0,Y 645.099,Z 1141.552,A -85,B 0,C 180,E1 5835.886,E2 5835.886} C_VEL
LIN {X 0,Y 643.577,Z 1171.664,A -85,B 0,C 180,E1 5841.851,E2 5841.851} C_VEL
LIN {X 0,Y 642.949,Z 1190.995,A -85,B 0,C 180,E1 5847.974,E2 5847.974} C_VEL
LIN {X 0,Y 643.089,Z 1199.031,A -85,B 0,C 180,E1 5853.382,E2 5853.382} C_VEL
LIN {X 0,Y 642.862,Z 1197.448,A -85,B 0,C 180,E1 5860.192,E2 5860.192} C_VEL
LIN {X 0,Y 643.044,Z 1184.456,A -85,B 0,C 180,E1 5866.441,E2 5866.441} C_VEL
LIN {X 0,Y 643.942,Z 1162.571,A -85,B 0,C 180,E1 5872.137,E2 5872.137} C_VEL
LIN {X 0,Y 646.004,Z 1127.022,A -85,B 0,C 180,E1 5878.266,E2 5878.266} C_VEL
LIN {X 0,Y 650.183,Z 1076.303,A -85,B 0,C 180,E1 5884.37,E2 5884.37} C_VEL
LIN {X 0,Y 656.054,Z 1013.128,A -85,B 0,C 180,E1 5889.71,E2 5889.71} C_VEL
LIN {X 0,Y 662.207,Z 943.841,A -85,B 0,C 180,E1 5893.711,E2 5893.711} C_VEL
LIN {X 0,Y 667.121,Z 870.331,A -85,B 0,C 180,E1 5896.405,E2 5896.405} C_VEL
LIN {X 0,Y 667.73,Z 811.873,A -85,B 0,C 180,E1 5897.725,E2 5897.725} C_VEL
LIN {X 0,Y 642.233,Z 767.06,A -85,B 0,C 180,E1 5900.638,E2 5900.638} C_VEL
LIN {X 0,Y 642.479,Z 767.06,A -85,B 0,C 180,E1 5909.491,E2 5909.491} C_VEL
LIN {X 0,Y 642.62,Z 767.06,A -85,B 0,C 180,E1 5918.773,E2 5918.773} C_VEL
LIN {X 0,Y 643.315,Z 767.06,A -85,B 0,C 180,E1 5928.04,E2 5928.04} C_VEL
LIN {X 0,Y 643.187,Z 767.06,A -85,B 0,C 180,E1 5937.959,E2 5937.959} C_VEL
LIN {X 0,Y 642.79,Z 767.06,A -85,B 0,C 180,E1 5946.082,E2 5946.082} C_VEL
LIN {X 0,Y 642.499,Z 767.06,A -85,B 0,C 180,E1 5954.339,E2 5954.339} C_VEL
LIN {X 0,Y 642.156,Z 767.06,A -85,B 0,C 180,E1 5962.924,E2 5962.924} C_VEL
LIN {X 0,Y 642.284,Z 767.06,A -85,B 0,C 180,E1 5970.499,E2 5970.499} C_VEL
LIN {X 0,Y 641.881,Z 767.06,A -85,B 0,C 180,E1 5979.178,E2 5979.178} C_VEL
LIN {X 0,Y 633.817,Z 767.06,A -85,B 0,C 180,E1 5982.29,E2 5982.29} C_VEL
LIN {X 0,Y 634.509,Z 768.9,A -85,B 0,C 180,E1 5984.654,E2 5984.654} C_VEL
LIN {X 0,Y 663.385,Z 822.533,A -85,B 0,C 180,E1 5987.907,E2 5987.907} C_VEL
LIN {X 0,Y 659.264,Z 901.365,A -85,B 0,C 180,E1 5989.7,E2 5989.7} C_VEL
LIN {X 0,Y 653.392,Z 976.95,A -85,B 0,C 180,E1 5992.963,E2 5992.963} C_VEL
LIN {X 0,Y 646.951,Z 1045.653,A -85,B 0,C 180,E1 5997.552,E2 5997.552} C_VEL
LIN {X 0,Y 641.551,Z 1103.632,A -85,B 0,C 180,E1 6003.122,E2 6003.122} C_VEL
LIN {X 0,Y 637.831,Z 1151.301,A -85,B 0,C 180,E1 6009.65,E2 6009.65} C_VEL
LIN {X 0,Y 635.682,Z 1184.855,A -85,B 0,C 180,E1 6016.548,E2 6016.548} C_VEL
LIN {X 0,Y 635.044,Z 1203.52,A -85,B 0,C 180,E1 6023.141,E2 6023.141} C_VEL
LIN {X 0,Y 635.273,Z 1209.402,A -85,B 0,C 180,E1 6027.946,E2 6027.946} C_VEL
LIN {X 0,Y 635.103,Z 1206.815,A -85,B 0,C 180,E1 6034.792,E2 6034.792} C_VEL
LIN {X 0,Y 635.256,Z 1193.304,A -85,B 0,C 180,E1 6041.008,E2 6041.008} C_VEL
LIN {X 0,Y 636.336,Z 1167.936,A -85,B 0,C 180,E1 6047.329,E2 6047.329} C_VEL
LIN {X 0,Y 638.776,Z 1130.474,A -85,B 0,C 180,E1 6053.529,E2 6053.529} C_VEL
LIN {X 0,Y 643.534,Z 1078.29,A -85,B 0,C 180,E1 6059.569,E2 6059.569} C_VEL
LIN {X 0,Y 650.045,Z 1013.995,A -85,B 0,C 180,E1 6064.782,E2 6064.782} C_VEL
LIN {X 0,Y 656.506,Z 943.528,A -85,B 0,C 180,E1 6068.66,E2 6068.66} C_VEL
LIN {X 0,Y 661.459,Z 869.371,A -85,B 0,C 180,E1 6071.195,E2 6071.195} C_VEL
LIN {X 0,Y 662.02,Z 815.759,A -85,B 0,C 180,E1 6072.312,E2 6072.312} C_VEL
LIN {X 0,Y 634.073,Z 767.06,A -85,B 0,C 180,E1 6075.581,E2 6075.581} C_VEL
LIN {X 0,Y 634.579,Z 767.06,A -85,B 0,C 180,E1 6084.169,E2 6084.169} C_VEL
LIN {X 0,Y 634.51,Z 767.06,A -85,B 0,C 180,E1 6092.23,E2 6092.23} C_VEL
LIN {X 0,Y 634.618,Z 767.06,A -85,B 0,C 180,E1 6101.19,E2 6101.19} C_VEL
LIN {X 0,Y 634.658,Z 767.06,A -85,B 0,C 180,E1 6111.077,E2 6111.077} C_VEL
LIN {X 0,Y 635.133,Z 767.06,A -85,B 0,C 180,E1 6117.961,E2 6117.961} C_VEL
LIN {X 0,Y 634.825,Z 767.06,A -85,B 0,C 180,E1 6126.186,E2 6126.186} C_VEL
LIN {X 0,Y 634.458,Z 767.06,A -85,B 0,C 180,E1 6134.553,E2 6134.553} C_VEL
LIN {X 0,Y 634.117,Z 767.06,A -85,B 0,C 180,E1 6142.976,E2 6142.976} C_VEL
LIN {X 0,Y 634.104,Z 767.06,A -85,B 0,C 180,E1 6150.967,E2 6150.967} C_VEL
LIN {X 0,Y 633.964,Z 767.06,A -85,B 0,C 180,E1 6159.368,E2 6159.368} C_VEL
LIN {X 0,Y 634.209,Z 767.06,A -85,B 0,C 180,E1 6167.045,E2 6167.045} C_VEL
LIN {X 0,Y 634.478,Z 768.928,A -85,B 0,C 180,E1 6170.76,E2 6170.76} C_VEL
LIN {X 0,Y 662.948,Z 821.004,A -85,B 0,C 180,E1 6173.974,E2 6173.974} C_VEL
LIN {X 0,Y 659.171,Z 896.263,A -85,B 0,C 180,E1 6175.838,E2 6175.838} C_VEL
LIN {X 0,Y 653.311,Z 969.443,A -85,B 0,C 180,E1 6179.066,E2 6179.066} C_VEL
LIN {X 0,Y 646.755,Z 1037.199,A -85,B 0,C 180,E1 6183.63,E2 6183.63} C_VEL
LIN {X 0,Y 641.125,Z 1095.841,A -85,B 0,C 180,E1 6189.319,E2 6189.319} C_VEL
LIN {X 0,Y 637.273,Z 1142.028,A -85,B 0,C 180,E1 6195.709,E2 6195.709} C_VEL
LIN {X 0,Y 635.606,Z 1172.321,A -85,B 0,C 180,E1 6201.841,E2 6201.841} C_VEL
LIN {X 0,Y 634.957,Z 1191.163,A -85,B 0,C 180,E1 6207.949,E2 6207.949} C_VEL
LIN {X 0,Y 635.069,Z 1199.084,A -85,B 0,C 180,E1 6213.424,E2 6213.424} C_VEL
LIN {X 0,Y 634.858,Z 1197.349,A -85,B 0,C 180,E1 6220.322,E2 6220.322} C_VEL
LIN {X 0,Y 635.087,Z 1184.335,A -85,B 0,C 180,E1 6226.615,E2 6226.615} C_VEL
LIN {X 0,Y 636,Z 1162.158,A -85,B 0,C 180,E1 6232.429,E2 6232.429} C_VEL
LIN {X 0,Y 638.286,Z 1127.045,A -85,B 0,C 180,E1 6238.547,E2 6238.547} C_VEL
LIN {X 0,Y 642.753,Z 1076.782,A -85,B 0,C 180,E1 6244.677,E2 6244.677} C_VEL
LIN {X 0,Y 648.934,Z 1014.888,A -85,B 0,C 180,E1 6249.991,E2 6249.991} C_VEL
LIN {X 0,Y 655.471,Z 946.572,A -85,B 0,C 180,E1 6254.016,E2 6254.016} C_VEL
LIN {X 0,Y 660.69,Z 873.735,A -85,B 0,C 180,E1 6256.768,E2 6256.768} C_VEL
LIN {X 0,Y 661.728,Z 815.359,A -85,B 0,C 180,E1 6258.13,E2 6258.13} C_VEL
LIN {X 0,Y 634.331,Z 767.06,A -85,B 0,C 180,E1 6261.376,E2 6261.376} C_VEL
LIN {X 0,Y 634.444,Z 767.06,A -85,B 0,C 180,E1 6270.746,E2 6270.746} C_VEL
LIN {X 0,Y 634.418,Z 767.06,A -85,B 0,C 180,E1 6279.701,E2 6279.701} C_VEL
LIN {X 0,Y 635.356,Z 767.06,A -85,B 0,C 180,E1 6288.278,E2 6288.278} C_VEL
LIN {X 0,Y 635.188,Z 767.06,A -85,B 0,C 180,E1 6297.933,E2 6297.933} C_VEL
LIN {X 0,Y 634.748,Z 767.06,A -85,B 0,C 180,E1 6306.16,E2 6306.16} C_VEL
LIN {X 0,Y 634.444,Z 767.06,A -85,B 0,C 180,E1 6314.525,E2 6314.525} C_VEL
LIN {X 0,Y 634.148,Z 767.06,A -85,B 0,C 180,E1 6322.972,E2 6322.972} C_VEL
LIN {X 0,Y 634.167,Z 767.06,A -85,B 0,C 180,E1 6330.932,E2 6330.932} C_VEL
LIN {X 0,Y 633.889,Z 767.06,A -85,B 0,C 180,E1 6339.338,E2 6339.338} C_VEL
LIN {X 0,Y 633.817,Z 767.06,A -85,B 0,C 180,E1 6342.29,E2 6342.29} C_VEL
LIN {X 0,Y 626.13,Z 767.06,A -85,B 0,C 180,E1 6343.68,E2 6343.68} C_VEL
LIN {X 0,Y 657.43,Z 824.538,A -85,B 0,C 180,E1 6347.472,E2 6347.472} C_VEL
LIN {X 0,Y 652.924,Z 903.803,A -85,B 0,C 180,E1 6349.322,E2 6349.322} C_VEL
LIN {X 0,Y 646.572,Z 979.588,A -85,B 0,C 180,E1 6352.67,E2 6352.67} C_VEL
LIN {X 0,Y 639.714,Z 1047.504,A -85,B 0,C 180,E1 6357.301,E2 6357.301} C_VEL
LIN {X 0,Y 633.94,Z 1105.233,A -85,B 0,C 180,E1 6362.965,E2 6362.965} C_VEL
LIN {X 0,Y 629.962,Z 1152.386,A -85,B 0,C 180,E1 6369.569,E2 6369.569} C_VEL
LIN {X 0,Y 627.814,Z 1184.854,A -85,B 0,C 180,E1 6376.376,E2 6376.376} C_VEL
LIN {X 0,Y 627.079,Z 1203.52,A -85,B 0,C 180,E1 6383.053,E2 6383.053} C_VEL
LIN {X 0,Y 626.74,Z 1209.837,A -85,B 0,C 180,E1 6389.305,E2 6389.305} C_VEL
LIN {X 0,Y 626.917,Z 1205.886,A -85,B 0,C 180,E1 6395.55,E2 6395.55} C_VEL
LIN {X 0,Y 627.212,Z 1191.055,A -85,B 0,C 180,E1 6401.857,E2 6401.857} C_VEL
LIN {X 0,Y 628.563,Z 1164.76,A -85,B 0,C 180,E1 6408.204,E2 6408.204} C_VEL
LIN {X 0,Y 631.6,Z 1125.579,A -85,B 0,C 180,E1 6414.503,E2 6414.503} C_VEL
LIN {X 0,Y 636.923,Z 1071.574,A -85,B 0,C 180,E1 6420.596,E2 6420.596} C_VEL
LIN {X 0,Y 644.093,Z 1005.698,A -85,B 0,C 180,E1 6425.766,E2 6425.766} C_VEL
LIN {X 0,Y 650.879,Z 935.91,A -85,B 0,C 180,E1 6429.44,E2 6429.44} C_VEL
LIN {X 0,Y 655.758,Z 864.504,A -85,B 0,C 180,E1 6431.769,E2 6431.769} C_VEL
LIN {X 0,Y 656.096,Z 818.955,A -85,B 0,C 180,E1 6432.732,E2 6432.732} C_VEL
LIN {X 0,Y 626.022,Z 767.06,A -85,B 0,C 180,E1 6436.345,E2 6436.345} C_VEL
LIN {X 0,Y 626.576,Z 767.06,A -85,B 0,C 180,E1 6445.343,E2 6445.343} C_VEL
LIN {X 0,Y 626.483,Z 767.06,A -85,B 0,C 180,E1 6453.405,E2 6453.405} C_VEL
LIN {X 0,Y 626.548,Z 767.06,A -85,B 0,C 180,E1 6462.94,E2 6462.94} C_VEL
LIN {X 0,Y 626.661,Z 767.06,A -85,B 0,C 180,E1 6470.962,E2 6470.962} C_VEL
LIN {X 0,Y 627.153,Z 767.06,A -85,B 0,C 180,E1 6477.935,E2 6477.935} C_VEL
LIN {X 0,Y 626.794,Z 767.06,A -85,B 0,C 180,E1 6486.266,E2 6486.266} C_VEL
LIN {X 0,Y 626.391,Z 767.06,A -85,B 0,C 180,E1 6494.744,E2 6494.744} C_VEL
LIN {X 0,Y 626.267,Z 767.06,A -85,B 0,C 180,E1 6502.065,E2 6502.065} C_VEL
LIN {X 0,Y 626.125,Z 767.06,A -85,B 0,C 180,E1 6510.71,E2 6510.71} C_VEL
LIN {X 0,Y 626.08,Z 767.06,A -85,B 0,C 180,E1 6518.174,E2 6518.174} C_VEL
LIN {X 0,Y 626.211,Z 767.06,A -85,B 0,C 180,E1 6526.359,E2 6526.359} C_VEL
LIN {X 0,Y 626.357,Z 768.823,A -85,B 0,C 180,E1 6530.005,E2 6530.005} C_VEL
LIN {X 0,Y 656.927,Z 821.772,A -85,B 0,C 180,E1 6533.514,E2 6533.514} C_VEL
LIN {X 0,Y 652.848,Z 898.317,A -85,B 0,C 180,E1 6535.45,E2 6535.45} C_VEL
LIN {X 0,Y 646.573,Z 970.844,A -85,B 0,C 180,E1 6538.703,E2 6538.703} C_VEL
LIN {X 0,Y 639.601,Z 1038.093,A -85,B 0,C 180,E1 6543.302,E2 6543.302} C_VEL
LIN {X 0,Y 633.595,Z 1096.543,A -85,B 0,C 180,E1 6549.061,E2 6549.061} C_VEL
LIN {X 0,Y 629.468,Z 1142.504,A -85,B 0,C 180,E1 6555.528,E2 6555.528} C_VEL
LIN {X 0,Y 627.705,Z 1172.353,A -85,B 0,C 180,E1 6561.667,E2 6561.667} C_VEL
LIN {X 0,Y 626.981,Z 1191.331,A -85,B 0,C 180,E1 6567.923,E2 6567.923} C_VEL
LIN {X 0,Y 627.049,Z 1199.138,A -85,B 0,C 180,E1 6573.468,E2 6573.468} C_VEL
LIN {X 0,Y 626.854,Z 1197.251,A -85,B 0,C 180,E1 6580.455,E2 6580.455} C_VEL
LIN {X 0,Y 627.107,Z 1184.653,A -85,B 0,C 180,E1 6586.643,E2 6586.643} C_VEL
LIN {X 0,Y 628.135,Z 1161.752,A -85,B 0,C 180,E1 6592.725,E2 6592.725} C_VEL
LIN {X 0,Y 630.632,Z 1126.073,A -85,B 0,C 180,E1 6598.986,E2 6598.986} C_VEL
LIN {X 0,Y 635.391,Z 1076.768,A -85,B 0,C 180,E1 6605.044,E2 6605.044} C_VEL
LIN {X 0,Y 642.234,Z 1013.675,A -85,B 0,C 180,E1 6610.494,E2 6610.494} C_VEL
LIN {X 0,Y 649.164,Z 945.25,A -85,B 0,C 180,E1 6614.528,E2 6614.528} C_VEL
LIN {X 0,Y 654.721,Z 872.851,A -85,B 0,C 180,E1 6617.25,E2 6617.25} C_VEL
LIN {X 0,Y 655.621,Z 818.612,A -85,B 0,C 180,E1 6618.557,E2 6618.557} C_VEL
LIN {X 0,Y 626.309,Z 767.06,A -85,B 0,C 180,E1 6621.949,E2 6621.949} C_VEL
LIN {X 0,Y 626.387,Z 767.06,A -85,B 0,C 180,E1 6630.22,E2 6630.22} C_VEL
LIN {X 0,Y 626.417,Z 767.06,A -85,B 0,C 180,E1 6639.43,E2 6639.43} C_VEL
LIN {X 0,Y 627.368,Z 767.06,A -85,B 0,C 180,E1 6648.234,E2 6648.234} C_VEL
LIN {X 0,Y 627.207,Z 767.06,A -85,B 0,C 180,E1 6657.907,E2 6657.907} C_VEL
LIN {X 0,Y 626.72,Z 767.06,A -85,B 0,C 180,E1 6666.239,E2 6666.239} C_VEL
LIN {X 0,Y 626.38,Z 767.06,A -85,B 0,C 180,E1 6674.716,E2 6674.716} C_VEL
LIN {X 0,Y 626.316,Z 767.06,A -85,B 0,C 180,E1 6682.033,E2 6682.033} C_VEL
LIN {X 0,Y 626.193,Z 767.06,A -85,B 0,C 180,E1 6690.712,E2 6690.712} C_VEL
LIN {X 0,Y 625.998,Z 767.06,A -85,B 0,C 180,E1 6698.145,E2 6698.145} C_VEL
LIN {X 0,Y 626.13,Z 767.06,A -85,B 0,C 180,E1 6703.68,E2 6703.68} C_VEL
LIN {X 0,Y 628.3,Z 775.797,A -85,B 0,C 180,E1 6704.192,E2 6704.192} C_VEL
LIN {X 0,Y 630.306,Z 788.536,A -85,B 0,C 180,E1 6704.58,E2 6704.58} C_VEL
LIN {X 0,Y 651.455,Z 828.214,A -85,B 0,C 180,E1 6707.053,E2 6707.053} C_VEL
